Universal Robots URScript: Floor Corner Extended.script

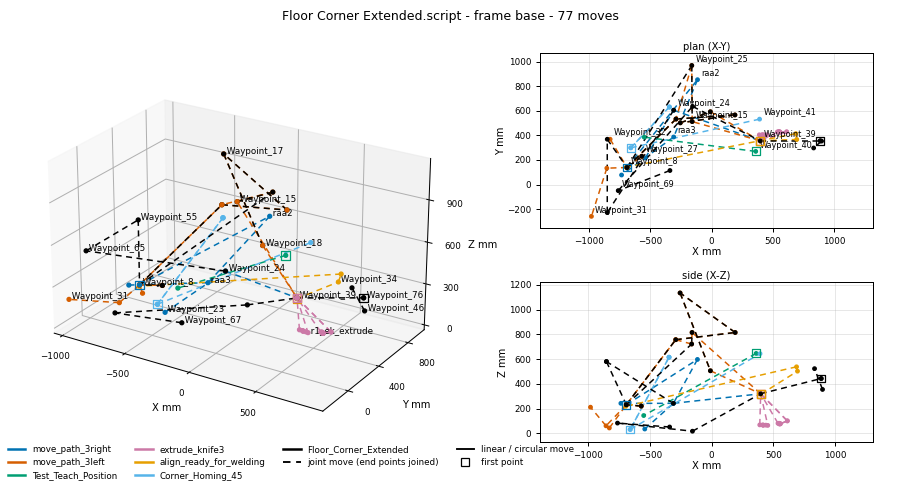
[picture p0: tool path of Floor Corner Extended.script in frame base, 77 of 152 moves have a stored position in this frame; points joined in program order, loops and branches not executed]
def Floor_Corner_Extended():
  global _hidden_verificationVariable=0
  step_count_477d2b75_14a1_4bd1_8ed8_9c73e5511d13 = 0.0
  thread Step_Counter_Thread_391a7927_408d_45dc_aa4e_0d8bac6dafc5():
    while (True):
      step_count_477d2b75_14a1_4bd1_8ed8_9c73e5511d13 = step_count_477d2b75_14a1_4bd1_8ed8_9c73e5511d13 + 1.0
      sync()
    end
  end
  run Step_Counter_Thread_391a7927_408d_45dc_aa4e_0d8bac6dafc5()
  set_tool_communication(False, 115200, 0, 1, 1.5, 3.5)
  set_tool_output_mode(0)
  set_tool_digital_output_mode(0, 1)
  set_tool_digital_output_mode(1, 1)
  set_tool_voltage(0)
  set_tcp(p[1.4000000000000001E-4,-0.01751,0.284,0.0,0.0,0.0])
  set_target_payload(10.800000, [-0.001000, -0.053000, 0.068000], [0.081228, 0.081228, 0.081228, 0.000000, 0.000000, 0.000000])
  set_gravity([0.0, 0.0, 9.82])
  set_standard_analog_input_domain(0, 1)
  set_standard_analog_input_domain(1, 1)
  set_tool_analog_input_domain(0, 1)
  set_tool_analog_input_domain(1, 1)
  set_analog_outputdomain(0, 0)
  set_analog_outputdomain(1, 0)
  set_input_actions_to_default()
  set_safety_mode_transition_hardness(1)
  global robot_number=2
  global Point_1=p[0.0,0.0,0.0,0.0,0.0,0.0]
  global Point_2=p[0.0,0.0,0.0,0.0,0.0,0.0]
  # begin: URCap Installation Node
  #   Source: UR Connect, 1.13.79, Universal Robots
  #   Type: UR Connect
  myurRPC = rpc_factory("xmlrpc","http://127.0.0.1:40474")
  # end: URCap Installation Node
  # begin: URCap Installation Node
  #   Source: MachineLogic for Universal Robots, 3.1.7, Vention Inc.
  #   Type: MachineLogic for Universal Robots
  def waitForResponse(expected_response_vention, cname_vention):
  response_vention = socket_read_string(cname_vention,timeout=15)
  while response_vention != expected_response_vention:
  sleep(0.01)
  response_vention = socket_read_string(cname_vention,timeout=15)
  end
  sleep(0.01)
  sync()
  end
  def sendString(string_vention, expected_response_vention, cname_vention):
  socket_send_string(str_cat(string_vention,";"), cname_vention)
  response_vention = socket_read_string(cname_vention,timeout=15)
  if(response_vention == "nAck"):
  popup("nAck received")
  end
  while response_vention != expected_response_vention:
  sleep(0.01)
  response_vention = socket_read_string(cname_vention,timeout=15)
  if(response_vention == "nAck"):
  popup("nAck received")
  end
  end
  sleep(0.01)
  sync()
  end
  def sendStringNAck(string_vention, expected_response_vention, cname_vention):
  socket_send_string(str_cat(string_vention,";"), cname_vention)
  response_vention = socket_read_string(cname_vention,timeout=15)
  if(response_vention == "nAck"):
  popup("nAck received")
  end
  while(response_vention != expected_response_vention and response_vention != "nAck"):
  sleep(0.01)
  response_vention = socket_read_string(cname_vention,timeout=15)
  if(response_vention == "nAck"):
  popup("nAck received",blocking=True)
  end
  end
  sleep(0.01)
  sync()
  end
  def sendStringWithTimeout(string_vention, expected_response_vention, cname_vention):
  socket_send_string(str_cat(string_vention,";"), cname_vention)
  response_vention = socket_read_string(cname_vention,timeout=10)
  if(response_vention == "nAck"):
  popup("nAck received"+string_vention)
  end
  sleep(0.01)
  sync()
  end
  def pollString(string_vention, expected_response_vention, cname_vention):
  socket_send_string(str_cat(string_vention,";"), cname_vention)
  response_vention = socket_read_string(cname_vention,timeout=15)
  if(response_vention == "nAck"):
  popup("nAck received")
  end
  while response_vention != expected_response_vention:
  sleep(1)
  socket_send_string(str_cat(string_vention,";"), cname_vention)
  response_vention = socket_read_string(cname_vention,timeout=15)
  if(response_vention == "nAck"):
  popup("nAck received")
  end
  end
  sleep(0.01)
  sync()
  end
  def sendVariable(var_vention, data_vention, expected_response_vention, cname_vention):
  socket_set_var(var_vention, data_vention, cname_vention)
  response_vention = socket_read_string(cname_vention,timeout=15)
  if(response_vention == "nAck"):
  popup("nAck received")
  end
  while response_vention != expected_response_vention:
  sleep(0.01)
  response_vention = socket_read_string(cname_vention,timeout=15)
  if(response_vention == "nAck"):
  popup("nAck received")
  end
  end
  sleep(0.01)
  sync()
  end
  def intToString(integer_vention,cname_vention):
  stringFix=""
  multiplier_vention123=1
  if integer_vention<0:
  stringFix="-"
  multiplier_vention123=-1
  end
  socket_set_var("GetString",integer_vention*multiplier_vention123,cname_vention)
  string_vention=""
  while string_vention=="":
  sleep(0.01)
  string_vention=socket_read_string(cname_vention,timeout=15)
  end
  sleep(0.01)
  sync()
  string_vention=stringFix+string_vention
  return string_vention
  end
  string_vention=""
  isVentionMovementBusy = False
  isVentionParallelMovementSendingScript = False
  ventionThreadHandle = 1
  isVentionMovementBusyMachineMotion1 = False
  isVentionParallelMovementSendingScriptMachineMotion1 = False
  socket_vention = socket_open("192.168.3.52", 9999, "MachineMotion1")
  if socket_vention==False:
  popup("Check configuration, can't connect to MachineMotion")
  end
  waitForResponse("MachineMotion connection established", "MachineMotion1")
  sendString("isReady", "MachineMotion isReady = true", "MachineMotion1")
  sendStringWithTimeout("setURCapVersion2", "setURCapVersion loaded", "MachineMotion1")
  sendString("SET speed_v2 1000000", "Ack", "MachineMotion1")
  sendString("SET acceleration_v2 100000", "Ack", "MachineMotion1")
  sendString("SET de_axis_1_microsteps_config 8", "Ack", "MachineMotion1")
  sendString("SET de_axis_1_mechanical_gain_config_v2 150000.0", "Ack", "MachineMotion1")
  sendString("SET de_axis_1_direction_config 1", "Ack", "MachineMotion1")
  sendString("SET de_axis_1_type_config Custom Actuator ", "Ack", "MachineMotion1")
  sendString("de_axis_1_config_exec", "Ack", "MachineMotion1")
  # end: URCap Installation Node
  # begin: URCap Installation Node
  #   Source: WireTank Serial, 4.9.0, WireTank, LLC
  #   Type: WireTank Serial
  WTSerialBridge = rpc_factory("xmlrpc","http://127.0.0.1:40511/RPC2")
  # end: URCap Installation Node
  global free_dr_already=  False
  global freedrive_m_var=  False
  global Waypoint_76_p=p[.886939072471, .356263001241, .442999104957, 2.316306590719, 2.057646408592, .074101958719]
  global Waypoint_76_q=[-3.2647881984118814, -1.2522049299371645, 1.5824044773896437, 0.9175786249801816, -0.008369636028316307, -1.3112608249927966]
  global Waypoint_50_p=p[-.568711442653, .230601791901, .220208834751, -1.519093932087, -.535128035721, .573965472012]
  global Waypoint_50_q=[-0.021522347127095998, -1.2794721287539979, 2.4323821703540247, 5.090870934515753, -2.2996109167682093, 1.533644199371338]
  global Waypoint_51_p=p[-.689649894186, .139001107022, .230693120258, -.852023156701, -1.645963115617, 1.645984943001]
  global Waypoint_51_q=[-1.1454814116107386, -1.5427037247321387, 2.8454700152026575, 4.979047852545538, -4.902958456669943, 1.5718834400177002]
  global Waypoint_52_p=p[-.160992057407, .970528182050, .722037363514, -.554955923310, .106486629259, .328544950173]
  global Waypoint_52_q=[-1.2978580633746546, -1.3217003357461472, 2.2583277861224573, 3.7025129038044433, -2.952825371419088, 0.9627944231033325]
  global Waypoint_53_p=p[-.157624488365, .513351401913, .815670293526, -.672704566373, -1.852329693545, -.055423312366]
  global Waypoint_53_q=[-2.7676661650287073, -1.8206430874266566, 2.312763277684347, 1.0122546392628173, -1.0765226523028772, -0.8102834860431116]
  global Waypoint_54_p=p[-.308528116178, .606080777007, .242371251996, -2.133736658076, .349438277129, 2.130953356703]
  global Waypoint_54_q=[-1.9617512861834925, -1.2994225782207032, 2.207935158406393, 0.745708628291748, 1.5955500602722168, 1.41863214969635]
  global Waypoint_65_p=p[-.850299549699, -.229060500451, .580194265918, -.066683564301, -1.566406749139, -.045536147896]
  global Waypoint_65_q=[0.11527767777442932, -1.206728772526123, 2.660132948552267, 3.2525827127644042, -4.69939905801882, -0.18521625200380498]
  global Waypoint_55_p=p[-.850295942693, .369353811615, .580190947871, -.066690142153, -1.566409865149, -.045506050424]
  global Waypoint_55_q=[-0.89636737505068, -1.198587493305542, 2.6061368624316614, 3.3119169908710937, -4.700617257748739, 0.826545238494873]
  global Waypoint_59_p=p[-.689650832419, .138973473550, .230700469426, -.851985360280, -1.645991124348, 1.645990580233]
  global Waypoint_59_q=[-1.1454528013812464, -1.5427289356342335, 2.8454795519458216, 4.979044186859884, -4.902960960065023, 1.5718833208084106]
  global Waypoint_71_p=p[-.289684660393, .534258475721, .757199031184, -.295236718653, -.653013693815, .389426431276]
  global Waypoint_71_q=[-1.3941848913775843, -1.6550847492613734, 2.7336130777942103, 4.156678839320801, -3.798194471989767, 1.7310842275619507]
  global Waypoint_58_p=p[.191120239889, .567518478899, .815512910186, -.135765364935, .396070873472, .208834263225]
  global Waypoint_58_q=[-1.651280705128805, -1.7712346516051234, 2.617981735860006, 3.3066598612019042, -2.656208101903097, 0.8563313484191895]
  global Waypoint_56_p=p[-.254568281661, .502958752129, 1.135400507516, -.261908057482, -.749714619963, 1.349050618455]
  global Waypoint_56_q=[-2.0344861189471644, -1.9012485943236292, 2.469647232686178, 2.2012061315723876, -1.1677187124835413, -0.5094392935382288]
  global Waypoint_57_p=p[-.009221327687, .593713365169, .505808930157, -1.424394189587, -2.344106819810, -.527597949261]
  global Waypoint_57_q=[-2.920837704335348, -1.9932075939574183, 2.3856611887561243, 0.6815890508839111, -0.5688460508929651, -1.1506975332843226]
  global Waypoint_67_p=p[-.339169194335, .114271165560, .051007401747, -.434162127311, 1.872717119498, -1.885153895998]
  global Waypoint_67_q=[-1.410516087208883, -0.9778240484050293, 2.47756010690798, -1.72361483196401, -0.3956816832171839, 1.808600902557373]
  global Waypoint_69_p=p[-.760826542313, -.049762698068, .082649581767, -1.026233921905, -1.612699318499, 1.547123897415]
  global Waypoint_69_q=[-0.22154647508730108, -1.118469015961029, 2.7561236063586634, -1.5568565337783475, -3.851987902318136, 1.559481143951416]
  global Waypoint_70_p=p[-.154414768496, .636923137577, .016979120256, -.302753655748, 1.486961848367, .122240024639]
  global Waypoint_70_q=[-1.1281922499286097, -1.0678585332683106, 2.4290812651263636, -2.7994214497008265, -1.6034835020648401, 1.7401196956634521]
  global Waypoint_49_p=p[.397354147848, .356263001249, .319808682466, 2.316306590727, 2.057646408591, .074101958728]
  global Waypoint_49_q=[-3.4579480330096644, -2.0568953953185023, 2.3266006151782435, -0.2270372670939942, -0.1993797461139124, -0.10534602800478154]
  global Waypoint_75_p=p[.886939072471, .356263001241, .442999104957, 2.316306590719, 2.057646408592, .074101958719]
  global Waypoint_75_q=[-3.2647881984118814, -1.2522049299371645, 1.5824044773896437, 0.9175786249801816, -0.008369636028316307, -1.3112608249927966]
  global Waypoint_46_p=p[.897631799353, .353934909904, .354805178378, 2.318109555057, 2.056931948624, .061383861333]
  global Waypoint_46_q=[-3.2637236754046843, -1.174605057840683, 1.6528332869159141, 1.0000695425220945, -0.0017340818988245132, -1.5358897417550086]
  global Waypoint_20_p=p[.833090611797, .298095916052, .522915034559, -2.069934341898, -1.817090229983, .262480162787]
  global Waypoint_20_q=[-3.3684676667627205, -1.191816195275802, 1.4015747865517827, 0.7519456332104983, -0.12742073350990069, -0.5504001287532203]
  global Waypoint_8_p=p[-.689650873132, .138963273545, .230691387978, -.851994598965, -1.645998530536, 1.646007616333]
  global Waypoint_8_q=[-0.9414032141314905, -1.501500443821289, 2.801856819783346, 4.981602895050802, -4.698942009602682, 1.571649193763733]
  global raa1_p=p[-.689643170661, .139073527807, .230690921608, -.852069296672, -1.645944888292, 1.645881185303]
  global raa1_q=[-1.1455705801593226, -1.5426994071206828, 2.8454588095294397, 4.979022520571508, -4.9029627482043665, 1.5718539953231812]
  global raa2_p=p[-.114157470946, .855108345894, .597477301975, -.505907028801, .325764798924, .388694870300]
  global raa2_q=[-1.2560303846942347, -1.339010552769043, 2.4151175657855433, 3.6540276247211914, -2.7377544085132044, 1.1360299587249756]
  global raa3_p=p[-.308547482234, .387797636904, .242407099860, 1.976327760240, .350206946999, -1.916000398832]
  global raa3_q=[-1.8931763807879847, -1.3096025747111817, 2.212959591542379, 0.7217818933674316, 1.639076590538025, 0.8125834465026855]
  global raa4_p=p[-.733576132099, .077690893520, .242409727900, 1.976419296976, .350069431278, -1.916084616091]
  global raa4_q=[-0.8909156958209437, -1.3431089532426377, 2.273750130330221, 0.7266384798237304, 1.5611975193023682, 1.8127720355987549]
  global Waypoint_23_p=p[-.540166575654, .215949141041, .034631452617, -1.505795438113, 1.057579835594, 1.573514753692]
  global Waypoint_23_q=[-0.46167117754091436, -1.1365486842444916, 2.508885685597555, 0.15223841249432368, 1.4952874183654785, 3.819530963897705]
  global Waypoint_24_p=p[-.308525559537, .606096497354, .242373144855, -2.133742737559, .349425192770, 2.130939839044]
  global Waypoint_24_q=[-1.8709262053119105, -1.2877716285041352, 2.192875687276022, 0.7510036665150146, 1.5878156423568726, 1.5091480016708374]
  global Waypoint_39_p=p[.397377312153, .356253310648, .319810281486, 2.316317670744, 2.057592854035, .074120023159]
  global Waypoint_39_q=[-3.4579551855670374, -2.0568958721556605, 2.3265963236438196, -0.22706706941638188, -0.19935590425600225, -0.10534030595888311]
  global Waypoint_37_p=p[.397366630181, .356258644196, .319813668943, 2.316299214281, 2.057614642521, .074125657910]
  global Waypoint_37_q=[-3.4579508940326136, -2.056904455224508, 2.3265963236438196, -0.2270481151393433, -0.19937020937074834, -0.10535222688783819]
  global Waypoint_15_p=p[-.157621040248, .513353603496, .815677694745, -.672699538592, -1.852318447516, -.055422773001]
  global Waypoint_15_q=[-2.770456854497091, -1.8207680187621058, 2.3065691629992884, 1.0170823770710449, -1.0767205397235315, -0.8071182409869593]
  global Waypoint_25_p=p[-.161036555831, .970524399959, .722042384791, -.554954311189, .106465018540, .328580879483]
  global Waypoint_25_q=[-1.3071630636798304, -1.3366777312806626, 2.2083633581744593, 3.7187773424335937, -2.9519384543048304, 0.9132363796234131]
  global Waypoint_72_p=p[-.289685725237, .534256396594, .757196155975, -.295237726329, -.653009715205, .389435972469]
  global Waypoint_72_q=[-1.394179646168844, -1.6550847492613734, 2.7336154619800013, 4.156686468715332, -3.7981911341296595, 1.731092095375061]
  global Waypoint_26_p=p[-.689650873132, .138963273545, .230691387978, -.851994598965, -1.645998530536, 1.646007616333]
  global Waypoint_26_q=[-0.9414032141314905, -1.501500443821289, 2.801856819783346, 4.981602895050802, -4.698942009602682, 1.571649193763733]
  global Waypoint_27_p=p[-.568724745609, .230601805298, .220208295176, -1.519097711196, -.535155391172, .573964121010]
  global Waypoint_27_q=[-0.04883271852602178, -1.2753942471793671, 2.4771457354175013, 5.041022258787908, -2.326899592076437, 1.532160997390747]
  global Waypoint_28_p=p[-.568724745609, .230601805298, .220208295176, -1.519097711196, -.535155391172, .573964121010]
  global Waypoint_28_q=[-0.04883271852602178, -1.2753942471793671, 2.4771457354175013, 5.041022258787908, -2.326899592076437, 1.532160997390747]
  global Waypoint_29_p=p[-.689650873132, .138963273545, .230691387978, -.851994598965, -1.645998530536, 1.646007616333]
  global Waypoint_29_q=[-0.9414032141314905, -1.501500443821289, 2.801856819783346, 4.981602895050802, -4.698942009602682, 1.571649193763733]
  global Waypoint_30_p=p[-.853851193668, .133266829906, .060418082908, -.274178222953, -2.359710051999, .046821166283]
  global Waypoint_30_q=[-0.608560864125387, -1.0122360748103638, 2.787060801182882, 3.7283646303364257, -4.940747324620382, 0.3777344226837158]
  global Waypoint_31_p=p[-.979398188272, -.259625449453, .211289397035, -.673010443572, -1.459355862765, -.640164958946]
  global Waypoint_31_q=[0.36968713998794556, -0.5732358259013672, 2.138303581868307, 3.1253925996967773, -4.70385724702944, -1.2100523153888147]
  global Waypoint_32_p=p[-.826865752305, .369357632284, .043113676955, .574997346548, -1.492225541214, .597128135378]
  global Waypoint_32_q=[-1.0355513731585901, -0.33930082738909917, 2.126244846974508, 2.9386045175739746, -4.711197797452108, 1.7860286235809326]
  global Waypoint_33_p=p[-.689650873132, .138963273545, .230691387978, -.851994598965, -1.645998530536, 1.646007616333]
  global Waypoint_33_q=[-0.9414032141314905, -1.501500443821289, 2.801856819783346, 4.981602895050802, -4.698942009602682, 1.571649193763733]
  global Waypoint_73_p=p[-.289671192632, .534275423553, .757232902417, -.295189983811, -.652980753171, .389398176275]
  global Waypoint_73_q=[-1.39418870607485, -1.65509094814443, 2.7335642019854944, 4.156684561366699, -3.7981610933886927, 1.731088399887085]
  global Waypoint_16_p=p[.191112811238, .567512170908, .815514010937, -.135771161622, .396053809900, .208825693369]
  global Waypoint_16_q=[-1.6536315123187464, -1.762029310266012, 2.6225650946246546, 3.2891055780598144, -2.6549678484546106, 0.8520665764808655]
  global Waypoint_17_p=p[-.254565633623, .502963426820, 1.135401557820, -.261910507478, -.749716086887, 1.349041636154]
  global Waypoint_17_q=[-2.035229508076803, -1.8928028545775355, 2.468372408543722, 2.19391576826062, -1.167032543812887, -0.5091407934771937]
  global Waypoint_18_p=p[-.009208376822, .593717720951, .505810027228, -1.424406033077, -2.344120510145, -.527630245278]
  global Waypoint_18_q=[-2.9172328154193323, -1.9945279560484828, 2.3804522196399134, 0.6930715280720214, -0.5671199003802698, -1.1566088835345667]
  global Waypoint_38_p=p[.397379749540, .356252016937, .319817140705, 2.316310534508, 2.057580214841, .074134378577]
  global Waypoint_38_q=[-3.457958761845724, -2.0569073162474574, 2.3265913168536585, -0.22705944002185063, -0.19935638109316045, -0.10534793535341436]
  global Waypoint_40_p=p[.360688403366, .270119715397, .646144746546, .057805349154, 2.125995180379, 2.134053153683]
  global Waypoint_40_q=[-3.4579489866839808, -2.0569035015501917, 2.3265796343432825, -0.22706706941638188, -0.1993501822101038, -0.10534793535341436]
  global Waypoint_2_p=p[-.548957282596, .386284559177, .143710178207, 1.570800598292, -.000025190822, .000004803470]
  global Waypoint_2_q=[-1.0516188780414026, -1.010990933781006, 2.1562450567828577, -1.143702046280243, -1.0526168982135218, -0.0017235914813440445]
  global r1_ek_oldhome_p=p[.397380247322, .356253634699, .319820846021, 2.316316320871, 2.057594704604, .074118471609]
  global r1_ek_oldhome_q=[-3.457949940358297, -2.056894441644186, 2.32658034959902, -0.2270551484874268, -0.19935208955873662, -0.10533696809877569]
  global r1_ek_extrude_p=p[.454852104155, .405448828659, .064015413765, 2.316807606413, 2.051392071696, .076664825947]
  global r1_ek_extrude_q=[-3.274653975163595, -1.5604325172356148, 2.467809502278463, -0.34438879907641606, -0.014281574879781544, -0.6303489843951624]
  global r1_ek_front_p=p[.439064809878, .405452261046, .065996139932, 2.316843937268, 2.051427632497, .076607106393]
  global r1_ek_front_q=[-3.280560557042257, -1.6287623844542445, 2.502561871205465, -0.47416289270434575, -0.019731823598043263, -0.4669149557696741]
  global r1_ek_middle_p=p[.419010105608, .404850828431, .065994665459, 2.309574128677, 2.044678176343, .089098333896]
  global r1_ek_middle_q=[-3.290863100682394, -1.70143522838735, 2.548208538685934, -0.589385525589325, -0.029501263295308888, -0.3372734228717249]
  global r1_ek_middle2_p=p[.417011768852, .405435328663, .065002627117, 2.316867113472, 2.051334925313, .076628493429]
  global r1_ek_middle2_q=[-3.289830032979147, -1.6934038601317347, 2.5445857683764856, -0.579618052845337, -0.028589550648824513, -0.33885270753969365]
  global r1_ek_bottom_p=p[.413071667620, .405431286494, .067999701073, 2.316819721954, 2.051304037200, .076688572349]
  global r1_ek_bottom_q=[-3.2916205565081995, -1.708447118798727, 2.5485368410693567, -0.5849895042232056, -0.03033763567079717, -0.32244998613466436]
  global r1_ek_end_p=p[.389998638281, .405443674081, .068004818811, 2.316851991921, 2.051367741778, .076612018685]
  global r1_ek_end_q=[-3.3030064741717737, -1.7640062771239222, 2.5831297079669397, -0.63420523822818, -0.04154044786562139, -0.2521465460406702]
  global r2_ek_oldhome_p=p[.397380247322, .356253634699, .319820846021, 2.316316320871, 2.057594704604, .074118471609]
  global r2_ek_oldhome_q=[-3.461132842686933, -2.062320779349874, 2.32916033290004, -0.21924456446492258, -0.20097883707844666, -0.11039879152527199]
  global r2_ek_extrude_p=p[.612885745678, .429305279732, .100477107124, 2.149994969793, 2.225764025207, .087353352584]
  global r2_ek_extrude_q=[-3.199475796455825, -1.4862854517875999, 2.263543898005424, -0.6928175084157413, -0.09183293866530295, -0.15653548683830643]
  global r2_ek_front_p=p[.556405415915, .429305279815, .076984362723, -2.170411249256, -2.268200695165, -.015853660170]
  global r2_ek_front_q=[-3.2029012478485694, -1.4943971905029905, 2.3176866046272355, -0.727203417516419, -0.10461513056100813, -0.1013922369747533]
  global r2_ek_middle_p=p[.550033970532, .429305279917, .076253920653, -2.170411249261, -2.268200695170, -.015853660159]
  global r2_ek_middle_q=[-3.2036200175167613, -1.5006788185274456, 2.326226188945654, -0.730095076239345, -0.10533288811000929, -0.10075548926859312]
  global r2_ek_bottom_p=p[.546594660555, .429305280025, .080868477599, -2.170411249265, -2.268200695174, -.015853660149]
  global r2_ek_bottom_q=[-3.204010221105431, -1.5099366263094405, 2.3272215014458872, -0.722096275899732, -0.10572512264357048, -0.10049057923478166]
  global r2_ek_end_p=p[.537335106646, .429305280055, .080868477459, -2.170411249266, -2.268200695175, -.015853660146]
  global r2_ek_end_q=[-3.205098875769389, -1.5204959829395506, 2.3387656715508855, -0.724001524008818, -0.10681294496314919, -0.09956563917089412]
  global oldhome_p=p[.397683836105, .356251384911, .315246899233, 2.316304177919, 2.057561756051, .074146544723]
  global oldhome_q=[-3.457960907612936, -2.0569125614561976, 2.326589886342184, -0.22707636774096684, -0.19935208955873662, -0.10534269014467412]
  global Waypoint_34_p=p[.695155464390, .367451880816, .502522491683, 2.093108370749, 1.857548644474, .308841595089]
  global Waypoint_34_q=[-3.249415699635641, -1.9387923679747523, 2.3226097265826624, 3.981850786800049, -0.05697328249086553, 1.5286790132522583]
  global Waypoint_35_p=p[.687527620967, .415165960724, .537921070000, 2.127101811831, 1.929915403723, .470130777221]
  global Waypoint_35_q=[-3.249424997960226, -1.9387947521605433, 2.32263428369631, 3.9818588930317382, -6.198007937763826, 1.5286580324172974]
  global Waypoint_36_p=p[-.693756081485, .141369193308, .218584735520, -.851978179689, -1.646001533937, 1.646008371360]
  global Waypoint_36_q=[-1.1533568541156214, -1.4924076360515137, 2.8518698851214808, 4.922323781042852, -4.910887185727255, 1.5719373226165771]
  def calculate_point_to_move_towards(feature, direction, position_distance):
    local posDir=[direction[0], direction[1], direction[2]]
    if (norm(posDir) < 1e-6):
      return get_target_waypoint()
    end
    local direction_vector_normalized=normalize(posDir)
    local displacement_pose=p[direction_vector_normalized[0] * position_distance,direction_vector_normalized[1] * position_distance,direction_vector_normalized[2] * position_distance,0,0,0]
    local wanted_displacement_in_base_frame=pose_sub(pose_trans(feature, displacement_pose), feature)
    return pose_add(get_target_waypoint(), wanted_displacement_in_base_frame)
  end
  global Waypoint_4_p=p[-.658264763546, .299530128456, .030909835036, .426821001551, -1.621505068649, .437070885767]
  global Waypoint_4_q=[-1.350241486226217, -0.9702387017062684, 2.492185179387228, -1.7834822140135707, -0.33723670641054326, 1.8489984273910522]
  global Waypoint_13_p=p[-.343952006273, .632142227752, .615174722549, -.025948978133, -.008794819136, -.567469912202]
  global Waypoint_13_q=[-1.350241486226217, -0.9702451390079041, 2.492171827946798, -3.0669099293150843, 1.575993537902832, 2.355180025100708]
  global Waypoint_1_p=p[-.343952006258, .632142227456, .615174722551, -.025016780489, .033118613186, -3.068519793995]
  global Waypoint_1_q=[-1.3432858302651205, -0.8819789687502322, 2.478150442072055, -3.1920490209023007, 1.5816449765089289, -0.1549241290366341]
  global Waypoint_14_p=p[-.343952006273, .632142227752, .615174722549, -.025948978133, -.008794819136, -.567469912202]
  global Waypoint_14_q=[-1.350241486226217, -0.9702451390079041, 2.492171827946798, -3.0669099293150843, 1.575993537902832, 2.355180025100708]
  global Waypoint_41_p=p[.392127936214, .533269017847, .644148583936, .057822570580, 2.125982462550, 2.134033989912]
  global Waypoint_41_q=[-3.4579578081714075, -2.0569120846190394, 2.3265841642962855, -0.22706885755572515, -0.1993349234210413, -0.10534984270204717]
  def move_path_3right():
    $ 136 "move_path_3right" "noBreak"
    $ 137 "'this is the path for Down, Over, then Back Around'"
    # 'this is the path for Down, Over, then Back Around'
    $ 138 "Comment"
    # Comment
    $ 147 "align_ready_for_welding()"
    align_ready_for_welding()
    $ 148 "Comment"
    # Comment
    $ 149 "Set"
    set_tcp(p[-0.011699999999999999,-0.328,0.105,1.2092,-1.2092,1.2092])
    $ 150 "p1≔pathturn[0]"
    global p1=pathturn[0]
    $ 151 "p2≔pathturn[1]"
    global p2=pathturn[1]
    $ 152 "p4≔pathturn[2]"
    global p4=pathturn[2]
    $ 153 "p5≔pathturn[3]"
    global p5=pathturn[3]
    $ 154 "pa1≔p[p1[0]+0.05,p1[1]+0.05,p1[2],p1[3],p1[4],p1[5]]"
    global pa1=p[p1[0]+0.05,p1[1]+0.05,p1[2],p1[3],p1[4],p1[5]]
    $ 155 "liftcolumnup"
    $ 156 "liftcolumnz≔liftcolumnzneeded"
    global liftcolumnz=liftcolumnzneeded
    $ 157 "If liftcolumnz>0"
    if (liftcolumnz>0):
      # begin: URCap Program Node
      #   Source: MachineLogic for Universal Robots, 3.1.7, Vention Inc.
      #   Type: MachineLogic for Universal Robots
      $ 158 "MachineLogic Move to Position"
      while isVentionMovementBusyMachineMotion1==True:
      sleep(0.05)
      end
      if(isVentionMovementBusyMachineMotion1 == False):
      isVentionMovementBusyMachineMotion1 = True
      socket_send_string("estop/status;", "MachineMotion1")
      temp_estop_var_vention = socket_read_string("MachineMotion1",timeout=15)
      while(temp_estop_var_vention=="estop/status true"):
      if temp_estop_var_vention=="estop/status true":
      sendStringWithTimeout("estop/systemreset/request","Ack estop/systemreset/request;","MachineMotion1")
      end
      socket_send_string("estop/status;", "MachineMotion1")
      temp_estop_var_vention = socket_read_string("MachineMotion1",timeout=15)
      if temp_estop_var_vention=="estop/status true":
      popup("MachineMotion in estop, make sure you have all emergency modules released manually. If you continue the system will try to reset MachineMotion automatically.",blocking=True)
      end
      end
      else:
      popup("resource is being used already: MachineMotion1")
      halt
      end
      sendString("SET speed_v2 3000000.000", "Ack", "MachineMotion1")
      sendString("SET acceleration_v2 50000.000", "Ack", "MachineMotion1")
      string_vention=intToString(liftcolumnz*1000,"MachineMotion1")
      sendString("SET de_move_abs_1 "+string_vention, "Ack", "MachineMotion1")
      sendString("de_move_abs_exec", "Ack", "MachineMotion1")
      isVentionParallelMovementSendingScriptMachineMotion1 = False
      pollString("isMotionCompleted", "MachineMotion isMotionCompleted = true", "MachineMotion1")
      isVentionMovementBusyMachineMotion1 = False
      sleep(0.03)
      # end: URCap Program Node
    end
    $ 159 "MoveJ"
    $ 160 "pa1" "breakAfter"
    movej(pa1, a=1.3962634015954636, v=0.3490658503988659)
    $ 161 "MoveL"
    $ 162 "p1" "breakAfter"
    movel(p1, a=0.2, v=0.05)
    $ 163 "Wait: 8.0"
    sleep(8.0)
    # begin: URCap Program Node
    #   Source: WireTank Serial, 4.9.0, WireTank, LLC
    #   Type: WireTank Serial
    $ 164 "Serial Bridge uR1"
    SerialResponse = WTSerialBridge.send_command("/dev/ttyUSB0",1200, 8, "None", "One", "None", 1000, "None", "None", [252,82,49], False)
    # end: URCap Program Node
    # begin: URCap Program Node
    #   Source: WireTank Serial, 4.9.0, WireTank, LLC
    #   Type: WireTank Serial
    $ 165 "Serial Bridge uR1"
    SerialResponse = WTSerialBridge.send_command("/dev/ttyUSB0",1200, 8, "None", "One", "None", 1000, "None", "None", [252,82,49], False)
    # end: URCap Program Node
    $ 166 "Wait: 1.0"
    sleep(1.0)
    $ 168 "Set DO[0]=On"
    set_standard_digital_out(0, True)
    $ 169 "MoveL"
    $ 170 "p2" "breakAfter"
    movel(p2, a=0.1, v=0.01)
    # begin: URCap Program Node
    #   Source: WireTank Serial, 4.9.0, WireTank, LLC
    #   Type: WireTank Serial
    $ 171 "Serial Bridge uR0"
    SerialResponse = WTSerialBridge.send_command("/dev/ttyUSB0",1200, 8, "None", "One", "None", 1000, "None", "None", [252,82,48], False)
    # end: URCap Program Node
    $ 172 "Wait: 0.5"
    sleep(0.5)
    $ 173 "Set DO[0]=Off"
    set_standard_digital_out(0, False)
    $ 174 "MoveL"
    $ 175 "p4" "breakAfter"
    movel(p4, a=0.01, v=0.12)
    # begin: URCap Program Node
    #   Source: WireTank Serial, 4.9.0, WireTank, LLC
    #   Type: WireTank Serial
    $ 176 "Serial Bridge uR1"
    SerialResponse = WTSerialBridge.send_command("/dev/ttyUSB0",1200, 8, "None", "One", "None", 1000, "None", "None", [252,82,49], False)
    # end: URCap Program Node
    # begin: URCap Program Node
    #   Source: WireTank Serial, 4.9.0, WireTank, LLC
    #   Type: WireTank Serial
    $ 177 "Serial Bridge uR1"
    SerialResponse = WTSerialBridge.send_command("/dev/ttyUSB0",1200, 8, "None", "One", "None", 1000, "None", "None", [252,82,49], False)
    # end: URCap Program Node
    $ 178 "Wait: 1.0"
    sleep(1.0)
    $ 180 "Set DO[0]=On"
    set_standard_digital_out(0, True)
    $ 181 "MoveL"
    $ 182 "p5" "breakAfter"
    movel(p5, a=0.1, v=0.01)
    # begin: URCap Program Node
    #   Source: WireTank Serial, 4.9.0, WireTank, LLC
    #   Type: WireTank Serial
    $ 183 "Serial Bridge uR0"
    SerialResponse = WTSerialBridge.send_command("/dev/ttyUSB0",1200, 8, "None", "One", "None", 1000, "None", "None", [252,82,48], False)
    # end: URCap Program Node
    $ 184 "Wait: 2.0"
    sleep(2.0)
    $ 185 "Set DO[0]=Off"
    set_standard_digital_out(0, False)
    $ 186 "Comment"
    # Comment
    $ 187 "pret1≔p[p5[0]+.1,p5[1],p5[2],p5[3],p5[4],p5[5]]"
    global pret1=p[p5[0]+.1,p5[1],p5[2],p5[3],p5[4],p5[5]]
    $ 188 "p_1≔pathturn[4]"
    global p_1=pathturn[4]
    $ 189 "p_2≔pathturn[5]"
    global p_2=pathturn[5]
    $ 190 "p_3≔pathturn[6]"
    global p_3=pathturn[6]
    $ 191 "p_4≔pathturn[7]"
    global p_4=pathturn[7]
    $ 192 "p_5≔pathturn[8]"
    global p_5=pathturn[8]
    $ 193 "p_preheat≔p[p_3[0]+.01,p_3[1],p_3[2],p_3[3],p_3[4],p_3[5]]"
    global p_preheat=p[p_3[0]+.01,p_3[1],p_3[2],p_3[3],p_3[4],p_3[5]]
    $ 194 "p_pre_ret≔p[p_1[0]+.03,p_1[1]+.03,p_1[2],p_1[3],p_1[4],p_1[5]]"
    global p_pre_ret=p[p_1[0]+.03,p_1[1]+.03,p_1[2],p_1[3],p_1[4],p_1[5]]
    $ 195 "p_pre_ret2≔p[p_3[0]+.1,p_3[1],p_3[2],p_3[3],p_3[4],p_3[5]]"
    global p_pre_ret2=p[p_3[0]+.1,p_3[1],p_3[2],p_3[3],p_3[4],p_3[5]]
    $ 196 "'twist'"
    # 'twist'
    $ 197 "MoveJ"
    $ 198 "pret1" "breakAfter"
    movej(pret1, a=1.3962634015954636, v=1.3962634015954636)
    $ 199 "Waypoint_8" "breakAfter"
    movej(get_inverse_kin(Waypoint_8_p, qnear=Waypoint_8_q), a=1.3962634015954636, v=1.0471975511965976)
    $ 201 "MoveJ"
    $ 202 "raa1" "breakAfter"
    movej(get_inverse_kin(raa1_p, qnear=raa1_q), a=1.3962634015954636, v=1.0471975511965976)
    $ 203 "raa2" "breakAfter"
    movej(get_inverse_kin(raa2_p, qnear=raa2_q), a=1.3962634015954636, v=1.0471975511965976)
    $ 204 "raa3" "breakAfter"
    movej(get_inverse_kin(raa3_p, qnear=raa3_q), a=1.3962634015954636, v=1.0471975511965976)
    $ 205 "raa4" "breakAfter"
    movej(get_inverse_kin(raa4_p, qnear=raa4_q), a=1.3962634015954636, v=1.0471975511965976)
    $ 207 "If liftcolumnz≠0.0"
    if (liftcolumnz != 0.0):
      # begin: URCap Program Node
      #   Source: MachineLogic for Universal Robots, 3.1.7, Vention Inc.
      #   Type: MachineLogic for Universal Robots
      $ 208 "MachineLogic Homing"
      while isVentionMovementBusyMachineMotion1==True:
      sleep(0.05)
      end
      if(isVentionMovementBusyMachineMotion1 == False):
      isVentionMovementBusyMachineMotion1 = True
      socket_send_string("estop/status;", "MachineMotion1")
      temp_estop_var_vention = socket_read_string("MachineMotion1",timeout=15)
      while(temp_estop_var_vention=="estop/status true"):
      if temp_estop_var_vention=="estop/status true":
      sendStringWithTimeout("estop/systemreset/request","Ack estop/systemreset/request;","MachineMotion1")
      end
      socket_send_string("estop/status;", "MachineMotion1")
      temp_estop_var_vention = socket_read_string("MachineMotion1",timeout=15)
      if temp_estop_var_vention=="estop/status true":
      popup("MachineMotion in estop, make sure you have all emergency modules released manually. If you continue the system will try to reset MachineMotion automatically.",blocking=True)
      end
      end
      else:
      popup("resource is being used already: MachineMotion1")
      halt
      end
      isVentionMovementBusyMachineMotion1 = True
      sendString("im_home_axis_1", "MachineMotion im_home_axis_1 = completed", "MachineMotion1")
      isVentionMovementBusyMachineMotion1 = False
      sendString("SET im_set_encoder_pos_aux_1 0.000", "Ack", "MachineMotion1")
      isVentionMovementBusyMachineMotion1 = False
      sleep(0.03)
      # end: URCap Program Node
    end
    $ 209 "'preheat'"
    # 'preheat'
    $ 212 "MoveL"
    $ 213 "p_pre_ret2" "breakAfter"
    movel(p_pre_ret2, a=1.2, v=0.25)
    $ 214 "p_preheat" "breakAfter"
    movel(p_preheat, a=1.2, v=0.25)
    $ 215 "Wait: 6.0"
    sleep(6.0)
    $ 216 "MoveL"
    $ 217 "p_pre_ret2" "breakAfter"
    movel(p_pre_ret2, a=1.2, v=0.25)
    $ 218 "p_pre_ret" "breakAfter"
    movel(p_pre_ret, a=1.2, v=0.25)
    $ 219 "Set"
    set_tcp(p[0.00451,-0.328,0.105,1.2092,-1.2092,1.2092])
    $ 220 "MoveL"
    $ 221 "p_1" "breakAfter"
    movel(p_1, a=1.2, v=0.05)
    # begin: URCap Program Node
    #   Source: WireTank Serial, 4.9.0, WireTank, LLC
    #   Type: WireTank Serial
    $ 222 "Serial Bridge uR1"
    SerialResponse = WTSerialBridge.send_command("/dev/ttyUSB0",1200, 8, "None", "One", "None", 1000, "None", "None", [252,82,49], False)
    # end: URCap Program Node
    # begin: URCap Program Node
    #   Source: WireTank Serial, 4.9.0, WireTank, LLC
    #   Type: WireTank Serial
    $ 223 "Serial Bridge uR1"
    SerialResponse = WTSerialBridge.send_command("/dev/ttyUSB0",1200, 8, "None", "One", "None", 1000, "None", "None", [252,82,49], False)
    # end: URCap Program Node
    $ 224 "Wait: 1.0"
    sleep(1.0)
    $ 225 "Set DO[0]=On"
    set_standard_digital_out(0, True)
    $ 227 "Wait: 1.0"
    sleep(1.0)
    $ 228 "MoveL"
    $ 229 "p_2" "breakAfter"
    movel(p_2, a=1.2, v=0.01)
    $ 230 "MoveP"
    $ 231 "CircleMove"
    $ 232 "p_3" "noBreak"

    $ 233 "p_4" "breakAfter"
    movec(p_3, p_4, a=0.01, v=5.0E-4, r=0.0, mode=1)
    $ 234 "MoveL"
    $ 235 "p_5" "breakAfter"
    movel(p_5, a=1.2, v=0.012)
    # begin: URCap Program Node
    #   Source: WireTank Serial, 4.9.0, WireTank, LLC
    #   Type: WireTank Serial
    $ 236 "Serial Bridge uR0"
    SerialResponse = WTSerialBridge.send_command("/dev/ttyUSB0",1200, 8, "None", "One", "None", 1000, "None", "None", [252,82,48], False)
    # end: URCap Program Node
    $ 237 "Wait: 2.0"
    sleep(2.0)
    $ 238 "Set DO[0]=Off"
    set_standard_digital_out(0, False)
    $ 239 "MoveL"
    $ 240 "Waypoint_23" "breakAfter"
    movel(Waypoint_23_p, a=1.2, v=0.25)
    $ 241 "MoveJ"
    $ 242 "Waypoint_24" "breakAfter"
    movej(get_inverse_kin(Waypoint_24_p, qnear=Waypoint_24_q), a=1.3962634015954636, v=1.0471975511965976)
    $ 243 "Waypoint_39" "breakAfter"
    movej(get_inverse_kin(Waypoint_39_p, qnear=Waypoint_39_q), a=1.3962634015954636, v=1.0471975511965976)
    $ 244 "'above waypoint is home'"
    # 'above waypoint is home'
  end
  def move_path_3left():
    $ 245 "move_path_3left" "noBreak"
    $ 246 "'this is the path for Down, Over, then Back Around'"
    # 'this is the path for Down, Over, then Back Around'
    $ 247 "Comment"
    # Comment
    $ 248 "MoveJ"
    $ 249 "Waypoint_37" "breakAfter"
    movej(get_inverse_kin(Waypoint_37_p, qnear=Waypoint_37_q), a=1.3962634015954636, v=1.0471975511965976)
    $ 250 "'above point is home'"
    # 'above point is home'
    $ 251 "liftcolumnup"
    $ 252 "liftcolumnz≔liftcolumnzneeded"
    global liftcolumnz=liftcolumnzneeded
    $ 253 "If liftcolumnz>0"
    if (liftcolumnz>0):
      # begin: URCap Program Node
      #   Source: MachineLogic for Universal Robots, 3.1.7, Vention Inc.
      #   Type: MachineLogic for Universal Robots
      $ 254 "MachineLogic Move to Position"
      while isVentionMovementBusyMachineMotion1==True:
      sleep(0.05)
      end
      if(isVentionMovementBusyMachineMotion1 == False):
      isVentionMovementBusyMachineMotion1 = True
      socket_send_string("estop/status;", "MachineMotion1")
      temp_estop_var_vention = socket_read_string("MachineMotion1",timeout=15)
      while(temp_estop_var_vention=="estop/status true"):
      if temp_estop_var_vention=="estop/status true":
      sendStringWithTimeout("estop/systemreset/request","Ack estop/systemreset/request;","MachineMotion1")
      end
      socket_send_string("estop/status;", "MachineMotion1")
      temp_estop_var_vention = socket_read_string("MachineMotion1",timeout=15)
      if temp_estop_var_vention=="estop/status true":
      popup("MachineMotion in estop, make sure you have all emergency modules released manually. If you continue the system will try to reset MachineMotion automatically.",blocking=True)
      end
      end
      else:
      popup("resource is being used already: MachineMotion1")
      halt
      end
      sendString("SET speed_v2 3000000.000", "Ack", "MachineMotion1")
      sendString("SET acceleration_v2 50000.000", "Ack", "MachineMotion1")
      string_vention=intToString(liftcolumnz*1000,"MachineMotion1")
      sendString("SET de_move_abs_1 "+string_vention, "Ack", "MachineMotion1")
      sendString("de_move_abs_exec", "Ack", "MachineMotion1")
      isVentionParallelMovementSendingScriptMachineMotion1 = False
      pollString("isMotionCompleted", "MachineMotion isMotionCompleted = true", "MachineMotion1")
      isVentionMovementBusyMachineMotion1 = False
      sleep(0.03)
      # end: URCap Program Node
    end
    $ 255 "Waypoint_15" "breakAfter"
    movej(get_inverse_kin(Waypoint_15_p, qnear=Waypoint_15_q), a=1.3962634015954636, v=1.0471975511965976)
    $ 256 "Waypoint_25" "breakAfter"
    movej(get_inverse_kin(Waypoint_25_p, qnear=Waypoint_25_q), a=1.3962634015954636, v=1.0471975511965976)
    $ 257 "Waypoint_72" "breakAfter"
    movej(get_inverse_kin(Waypoint_72_p, qnear=Waypoint_72_q), a=1.3962634015954636, v=1.0471975511965976)
    $ 258 "Waypoint_26" "breakAfter"
    movej(get_inverse_kin(Waypoint_26_p, qnear=Waypoint_26_q), a=1.3962634015954636, v=1.0471975511965976)
    $ 259 "Waypoint_27" "breakAfter"
    movej(get_inverse_kin(Waypoint_27_p, qnear=Waypoint_27_q), a=1.3962634015954636, v=1.0471975511965976)
    $ 264 "Comment"
    # Comment
    $ 265 "Set"
    set_tcp(p[-0.011699999999999999,-0.328,0.105,1.2092,-1.2092,1.2092])
    $ 266 "p1≔pathturn[0]"
    global p1=pathturn[0]
    $ 267 "p2≔pathturn[1]"
    global p2=pathturn[1]
    $ 268 "p4≔pathturn[2]"
    global p4=pathturn[2]
    $ 269 "p5≔pathturn[3]"
    global p5=pathturn[3]
    $ 270 "pa1≔p[p1[0]+0.05,p1[1]-0.05,p1[2],p1[3],p1[4],p1[5]]"
    global pa1=p[p1[0]+0.05,p1[1]-0.05,p1[2],p1[3],p1[4],p1[5]]
    $ 271 "MoveJ"
    $ 272 "pa1" "breakAfter"
    movej(pa1, a=1.3962634015954636, v=1.0471975511965976)
    $ 273 "MoveL"
    $ 274 "p1" "breakAfter"
    movel(p1, a=0.1, v=0.05)
    $ 275 "Wait: 8.0"
    sleep(8.0)
    # begin: URCap Program Node
    #   Source: WireTank Serial, 4.9.0, WireTank, LLC
    #   Type: WireTank Serial
    $ 276 "Serial Bridge uR1"
    SerialResponse = WTSerialBridge.send_command("/dev/ttyUSB0",1200, 8, "None", "One", "None", 1000, "None", "None", [252,82,49], False)
    # end: URCap Program Node
    # begin: URCap Program Node
    #   Source: WireTank Serial, 4.9.0, WireTank, LLC
    #   Type: WireTank Serial
    $ 277 "Serial Bridge uR1"
    SerialResponse = WTSerialBridge.send_command("/dev/ttyUSB0",1200, 8, "None", "One", "None", 1000, "None", "None", [252,82,49], False)
    # end: URCap Program Node
    $ 278 "Wait: 1.0"
    sleep(1.0)
    $ 280 "Set DO[0]=On"
    set_standard_digital_out(0, True)
    $ 281 "MoveL"
    $ 282 "p2" "breakAfter"
    movel(p2, a=0.1, v=0.01)
    # begin: URCap Program Node
    #   Source: WireTank Serial, 4.9.0, WireTank, LLC
    #   Type: WireTank Serial
    $ 283 "Serial Bridge uR0"
    SerialResponse = WTSerialBridge.send_command("/dev/ttyUSB0",1200, 8, "None", "One", "None", 1000, "None", "None", [252,82,48], False)
    # end: URCap Program Node
    $ 284 "Wait: 0.5"
    sleep(0.5)
    $ 285 "Set DO[0]=Off"
    set_standard_digital_out(0, False)
    $ 286 "MoveL"
    $ 287 "p4" "breakAfter"
    movel(p4, a=0.01, v=0.12)
    # begin: URCap Program Node
    #   Source: WireTank Serial, 4.9.0, WireTank, LLC
    #   Type: WireTank Serial
    $ 288 "Serial Bridge uR1"
    SerialResponse = WTSerialBridge.send_command("/dev/ttyUSB0",1200, 8, "None", "One", "None", 1000, "None", "None", [252,82,49], False)
    # end: URCap Program Node
    # begin: URCap Program Node
    #   Source: WireTank Serial, 4.9.0, WireTank, LLC
    #   Type: WireTank Serial
    $ 289 "Serial Bridge uR1"
    SerialResponse = WTSerialBridge.send_command("/dev/ttyUSB0",1200, 8, "None", "One", "None", 1000, "None", "None", [252,82,49], False)
    # end: URCap Program Node
    $ 290 "Wait: 1.0"
    sleep(1.0)
    $ 292 "Set DO[0]=On"
    set_standard_digital_out(0, True)
    $ 293 "MoveL"
    $ 294 "p5" "breakAfter"
    movel(p5, a=0.1, v=0.01)
    # begin: URCap Program Node
    #   Source: WireTank Serial, 4.9.0, WireTank, LLC
    #   Type: WireTank Serial
    $ 295 "Serial Bridge uR0"
    SerialResponse = WTSerialBridge.send_command("/dev/ttyUSB0",1200, 8, "None", "One", "None", 1000, "None", "None", [252,82,48], False)
    # end: URCap Program Node
    $ 296 "Wait: 2.0"
    sleep(2.0)
    $ 297 "Set DO[0]=Off"
    set_standard_digital_out(0, False)
    $ 298 "Comment"
    # Comment
    $ 299 "pret1≔p[p5[0]+.1,p5[1],p5[2],p5[3],p5[4],p5[5]]"
    global pret1=p[p5[0]+.1,p5[1],p5[2],p5[3],p5[4],p5[5]]
    $ 300 "p_1≔pathturn[4]"
    global p_1=pathturn[4]
    $ 301 "p_2≔pathturn[5]"
    global p_2=pathturn[5]
    $ 302 "p_3≔pathturn[6]"
    global p_3=pathturn[6]
    $ 303 "p_4≔pathturn[7]"
    global p_4=pathturn[7]
    $ 304 "p_5≔pathturn[8]"
    global p_5=pathturn[8]
    $ 305 "p_preheat≔p[p_3[0]+.01,p_3[1],p_3[2],p_3[3],p_3[4],p_3[5]]"
    global p_preheat=p[p_3[0]+.01,p_3[1],p_3[2],p_3[3],p_3[4],p_3[5]]
    $ 306 "p_pre_ret≔p[p_1[0]+.03,p_1[1]-.03,p_1[2],p_1[3],p_1[4],p_1[5]]"
    global p_pre_ret=p[p_1[0]+.03,p_1[1]-.03,p_1[2],p_1[3],p_1[4],p_1[5]]
    $ 307 "p_pre_ret2≔p[p_3[0]+.03,p_3[1],p_3[2],p_3[3],p_3[4],p_3[5]]"
    global p_pre_ret2=p[p_3[0]+.03,p_3[1],p_3[2],p_3[3],p_3[4],p_3[5]]
    $ 308 "MoveJ"
    $ 309 "pret1" "breakAfter"
    movej(pret1, a=1.3962634015954636, v=1.3962634015954636)
    $ 310 "Waypoint_28" "breakAfter"
    movej(get_inverse_kin(Waypoint_28_p, qnear=Waypoint_28_q), a=1.3962634015954636, v=1.3962634015954636)
    $ 311 "If liftcolumnz≠0.0"
    if (liftcolumnz != 0.0):
      # begin: URCap Program Node
      #   Source: MachineLogic for Universal Robots, 3.1.7, Vention Inc.
      #   Type: MachineLogic for Universal Robots
      $ 312 "MachineLogic Homing"
      while isVentionMovementBusyMachineMotion1==True:
      sleep(0.05)
      end
      if(isVentionMovementBusyMachineMotion1 == False):
      isVentionMovementBusyMachineMotion1 = True
      socket_send_string("estop/status;", "MachineMotion1")
      temp_estop_var_vention = socket_read_string("MachineMotion1",timeout=15)
      while(temp_estop_var_vention=="estop/status true"):
      if temp_estop_var_vention=="estop/status true":
      sendStringWithTimeout("estop/systemreset/request","Ack estop/systemreset/request;","MachineMotion1")
      end
      socket_send_string("estop/status;", "MachineMotion1")
      temp_estop_var_vention = socket_read_string("MachineMotion1",timeout=15)
      if temp_estop_var_vention=="estop/status true":
      popup("MachineMotion in estop, make sure you have all emergency modules released manually. If you continue the system will try to reset MachineMotion automatically.",blocking=True)
      end
      end
      else:
      popup("resource is being used already: MachineMotion1")
      halt
      end
      isVentionMovementBusyMachineMotion1 = True
      sendString("im_home_axis_1", "MachineMotion im_home_axis_1 = completed", "MachineMotion1")
      isVentionMovementBusyMachineMotion1 = False
      sendString("SET im_set_encoder_pos_aux_1 0.000", "Ack", "MachineMotion1")
      isVentionMovementBusyMachineMotion1 = False
      sleep(0.03)
      # end: URCap Program Node
    end
    $ 313 "'now go into the ccw weld position'"
    # 'now go into the ccw weld position'
    $ 314 "Waypoint_29" "breakAfter"
    movej(get_inverse_kin(Waypoint_29_p, qnear=Waypoint_29_q), a=1.3962634015954636, v=1.3962634015954636)
    $ 315 "Comment"
    # Comment
    $ 316 "Waypoint_30" "breakAfter"
    movej(get_inverse_kin(Waypoint_30_p, qnear=Waypoint_30_q), a=1.3962634015954636, v=1.3962634015954636)
    $ 317 "Waypoint_31" "breakAfter"
    movej(get_inverse_kin(Waypoint_31_p, qnear=Waypoint_31_q), a=1.3962634015954636, v=1.3962634015954636)
    $ 326 "MoveL"
    $ 327 "p_pre_ret" "breakAfter"
    movel(p_pre_ret, a=1.2, v=0.25)
    $ 328 "p_pre_ret2" "breakAfter"
    movel(p_pre_ret2, a=1.2, v=0.25)
    $ 329 "p_preheat" "breakAfter"
    movel(p_preheat, a=1.2, v=0.25)
    $ 330 "Wait: 6.0"
    sleep(6.0)
    $ 331 "MoveL"
    $ 332 "p_pre_ret2" "breakAfter"
    movel(p_pre_ret2, a=1.2, v=0.25)
    $ 333 "p_pre_ret" "breakAfter"
    movel(p_pre_ret, a=1.2, v=0.25)
    $ 334 "Set"
    set_tcp(p[0.00451,-0.328,0.105,1.2092,-1.2092,1.2092])
    $ 335 "MoveL"
    $ 336 "p_1" "breakAfter"
    movel(p_1, a=0.1, v=0.05)
    # begin: URCap Program Node
    #   Source: WireTank Serial, 4.9.0, WireTank, LLC
    #   Type: WireTank Serial
    $ 337 "Serial Bridge uR1"
    SerialResponse = WTSerialBridge.send_command("/dev/ttyUSB0",1200, 8, "None", "One", "None", 1000, "None", "None", [252,82,49], False)
    # end: URCap Program Node
    # begin: URCap Program Node
    #   Source: WireTank Serial, 4.9.0, WireTank, LLC
    #   Type: WireTank Serial
    $ 338 "Serial Bridge uR1"
    SerialResponse = WTSerialBridge.send_command("/dev/ttyUSB0",1200, 8, "None", "One", "None", 1000, "None", "None", [252,82,49], False)
    # end: URCap Program Node
    $ 339 "Wait: 1.0"
    sleep(1.0)
    $ 340 "Set DO[0]=On"
    set_standard_digital_out(0, True)
    $ 342 "Wait: 1.0"
    sleep(1.0)
    $ 343 "MoveL"
    $ 344 "p_2" "breakAfter"
    movel(p_2, a=1.2, v=0.01)
    $ 345 "MoveP"
    $ 346 "CircleMove"
    $ 347 "p_3" "noBreak"

    $ 348 "p_4" "breakAfter"
    movec(p_3, p_4, a=0.01, v=5.0E-4, r=0.0, mode=1)
    $ 349 "MoveL"
    $ 350 "p_5" "breakAfter"
    movel(p_5, a=1.2, v=0.012)
    # begin: URCap Program Node
    #   Source: WireTank Serial, 4.9.0, WireTank, LLC
    #   Type: WireTank Serial
    $ 351 "Serial Bridge uR0"
    SerialResponse = WTSerialBridge.send_command("/dev/ttyUSB0",1200, 8, "None", "One", "None", 1000, "None", "None", [252,82,48], False)
    # end: URCap Program Node
    $ 352 "Wait: 2.0"
    sleep(2.0)
    $ 353 "Set DO[0]=Off"
    set_standard_digital_out(0, False)
    $ 358 "MoveJ"
    $ 359 "Waypoint_32" "breakAfter"
    movej(get_inverse_kin(Waypoint_32_p, qnear=Waypoint_32_q), a=1.3962634015954636, v=1.0471975511965976)
    $ 360 "Waypoint_33" "breakAfter"
    movej(get_inverse_kin(Waypoint_33_p, qnear=Waypoint_33_q), a=1.3962634015954636, v=1.0471975511965976)
    $ 361 "Waypoint_73" "breakAfter"
    movej(get_inverse_kin(Waypoint_73_p, qnear=Waypoint_73_q), a=1.3962634015954636, v=1.0471975511965976)
    $ 362 "Comment"
    # Comment
    $ 363 "MoveJ"
    $ 364 "Waypoint_16" "breakAfter"
    movej(get_inverse_kin(Waypoint_16_p, qnear=Waypoint_16_q), a=1.3962634015954636, v=1.0471975511965976)
    $ 365 "Waypoint_17" "breakAfter"
    movej(get_inverse_kin(Waypoint_17_p, qnear=Waypoint_17_q), a=1.3962634015954636, v=1.0471975511965976)
    $ 366 "Waypoint_18" "breakAfter"
    movej(get_inverse_kin(Waypoint_18_p, qnear=Waypoint_18_q), a=1.3962634015954636, v=1.0471975511965976)
    $ 367 "Waypoint_38" "breakAfter"
    movej(get_inverse_kin(Waypoint_38_p, qnear=Waypoint_38_q), a=1.3962634015954636, v=1.0471975511965976)
    $ 368 "'above point is home'"
    # 'above point is home'
  end
  def Test_Teach_Position():
    $ 369 "Test_Teach_Position" "noBreak"
    $ 373 "MoveJ"
    $ 374 "Waypoint_40" "breakAfter"
    set_tcp(p[0.0,0.0,0.019,0.0,0.0,0.0])
    movej(get_inverse_kin(Waypoint_40_p, qnear=Waypoint_40_q), a=1.3962634015954636, v=1.0471975511965976)
    $ 375 "'above waypoint is home'"
    # 'above waypoint is home'
    $ 376 "Waypoint_2" "breakAfter"
    set_tcp(p[0.0,0.0,0.019,0.0,0.0,0.0])
    movej(get_inverse_kin(Waypoint_2_p, qnear=Waypoint_2_q), a=1.3962634015954636, v=1.0471975511965976)
    $ 377 "Set"
    set_tcp(p[1.4000000000000001E-4,-0.01751,0.284,0.0,0.0,0.0])
    $ 378 "freedrive_m_var≔ False "
    global freedrive_m_var=  False
    $ 379 "freedrive_m_var≔ True "
    global freedrive_m_var=  True
    $ 380 "Popup: Move the TCP to the top of the weld, then click 'Continue'"
    popup("Move the TCP to the top of the weld, then click 'Continue'", "Message", False, False, blocking=True)
    $ 381 "tcp_pose_top≔get_actual_tcp_pose()"
    global tcp_pose_top= get_actual_tcp_pose ()
    $ 382 "Popup: Move the TCP to the corner of the tank, then click 'Continue'"
    popup("Move the TCP to the corner of the tank, then click 'Continue'", "Message", False, False, blocking=True)
    $ 383 "tcp_pose≔get_actual_tcp_pose()"
    global tcp_pose= get_actual_tcp_pose ()
    $ 384 "freedrive_m_var≔ False "
    global freedrive_m_var=  False
    $ 385 "Wait: 0.25"
    sleep(0.25)
    $ 386 "sync()"
    sync()
  end
  def align_tcp_left():
    $ 387 "align_tcp_left" "noBreak"
    $ 388 "'this program aligns the tcp parallel to the y direction'"
    # 'this program aligns the tcp parallel to the y direction'
    $ 389 "cp≔get_actual_tcp_pose()"
    global cp= get_actual_tcp_pose ()
    $ 390 "aligned_y_pose≔p[cp[0],cp[1],cp[2],1.570796,0,0]"
    global aligned_y_pose=p[cp[0],cp[1],cp[2],1.570796,0,0]
    $ 391 "MoveJ"
    $ 392 "aligned_y_pose" "breakAfter"
    movej(aligned_y_pose, a=1.3962634015954636, v=1.0471975511965976)
  end
  def extrude_knife3():
    $ 393 "extrude_knife3" "noBreak"
    $ 394 "pre program stuff"
    $ 395 "Set"
    set_tcp(p[-0.011699999999999999,-0.328,0.105,1.2092,-1.2092,1.2092])
    $ 396 "ek_sp≔get_actual_tcp_pose()"
    global ek_sp= get_actual_tcp_pose ()
    $ 397 "MoveL"
    $ 398 "ek_sp" "breakAfter"
    movel(ek_sp, a=1.2, v=0.005)
    $ 399 "'list possible points'"
    # 'list possible points'
    $ 400 "robot 1 moves"
    $ 401 "If 1≟2"
    if (1 == 2):
      $ 402 "MoveJ"
      $ 403 "r1_ek_oldhome" "breakAfter"
      movej(get_inverse_kin(r1_ek_oldhome_p, qnear=r1_ek_oldhome_q), a=1.3962634015954636, v=1.0471975511965976)
      $ 404 "r1_ek_extrude" "breakAfter"
      movej(get_inverse_kin(r1_ek_extrude_p, qnear=r1_ek_extrude_q), a=1.3962634015954636, v=1.0471975511965976)
      $ 405 "r1_ek_front" "breakAfter"
      movej(get_inverse_kin(r1_ek_front_p, qnear=r1_ek_front_q), a=1.3962634015954636, v=1.0471975511965976)
      $ 406 "r1_ek_middle" "breakAfter"
      movej(get_inverse_kin(r1_ek_middle_p, qnear=r1_ek_middle_q), a=1.3962634015954636, v=1.0471975511965976)
      $ 407 "r1_ek_middle2" "breakAfter"
      movej(get_inverse_kin(r1_ek_middle2_p, qnear=r1_ek_middle2_q), a=1.3962634015954636, v=1.0471975511965976)
      $ 408 "r1_ek_bottom" "breakAfter"
      movej(get_inverse_kin(r1_ek_bottom_p, qnear=r1_ek_bottom_q), a=1.3962634015954636, v=1.0471975511965976)
      $ 409 "r1_ek_end" "breakAfter"
      movej(get_inverse_kin(r1_ek_end_p, qnear=r1_ek_end_q), a=1.3962634015954636, v=1.0471975511965976)
    end
    $ 410 "robot 2 moves"
    $ 411 "If 1≟2"
    if (1 == 2):
      $ 412 "MoveJ"
      $ 413 "r2_ek_oldhome" "breakAfter"
      movej(get_inverse_kin(r2_ek_oldhome_p, qnear=r2_ek_oldhome_q), a=1.3962634015954636, v=1.0471975511965976)
      $ 415 "r2_ek_extrude" "breakAfter"
      movej(get_inverse_kin(r2_ek_extrude_p, qnear=r2_ek_extrude_q), a=1.3962634015954636, v=1.0471975511965976)
      $ 416 "r2_ek_front" "breakAfter"
      movej(get_inverse_kin(r2_ek_front_p, qnear=r2_ek_front_q), a=1.3962634015954636, v=1.0471975511965976)
      $ 417 "r2_ek_middle" "breakAfter"
      movej(get_inverse_kin(r2_ek_middle_p, qnear=r2_ek_middle_q), a=1.3962634015954636, v=1.0471975511965976)
      $ 418 "r2_ek_bottom" "breakAfter"
      movej(get_inverse_kin(r2_ek_bottom_p, qnear=r2_ek_bottom_q), a=1.3962634015954636, v=1.0471975511965976)
      $ 419 "r2_ek_end" "breakAfter"
      movej(get_inverse_kin(r2_ek_end_p, qnear=r2_ek_end_q), a=1.3962634015954636, v=1.0471975511965976)
    end
    $ 420 "'detemine correct points for which robot'"
    # 'detemine correct points for which robot'
    $ 421 "If robot_number≟1"
    if (robot_number == 1):
      $ 422 "robot1 positions"
      $ 423 "ek_oldhome≔r1_ek_oldhome_p"
      global ek_oldhome=r1_ek_oldhome_p
      $ 424 "ek_extrude≔r1_ek_extrude_p"
      global ek_extrude=r1_ek_extrude_p
      $ 425 "ek_front≔r1_ek_front_p"
      global ek_front=r1_ek_front_p
      $ 426 "ek_middle≔r1_ek_middle_p"
      global ek_middle=r1_ek_middle_p
      $ 427 "ek_middle2≔r1_ek_middle2_p"
      global ek_middle2=r1_ek_middle2_p
      $ 428 "ek_bottom≔r1_ek_bottom_p"
      global ek_bottom=r1_ek_bottom_p
      $ 429 "ek_end≔r1_ek_end_q"
      global ek_end=r1_ek_end_q
    else:
      $ 430 "ElseIf robot_number≟2"
      if (robot_number == 2):
        $ 431 "robot1 positions"
        $ 432 "ek_oldhome≔r2_ek_oldhome_p"
        global ek_oldhome=r2_ek_oldhome_p
        $ 433 "ek_extrude≔r2_ek_extrude_p"
        global ek_extrude=r2_ek_extrude_p
        $ 434 "ek_front≔r2_ek_front_p"
        global ek_front=r2_ek_front_p
        $ 435 "ek_middle≔r2_ek_middle_p"
        global ek_middle=r2_ek_middle_p
        $ 436 "ek_middle2≔r2_ek_middle_p"
        global ek_middle2=r2_ek_middle_p
        $ 437 "ek_bottom≔r2_ek_bottom_p"
        global ek_bottom=r2_ek_bottom_p
        $ 438 "ek_end≔r2_ek_end_q"
        global ek_end=r2_ek_end_q
      end
    end
    $ 439 "'start of program'"
    # 'start of program'
    $ 441 "Set"
    set_tcp(p[-0.011699999999999999,-0.328,0.105,1.2092,-1.2092,1.2092])
    $ 442 "MoveJ"
    $ 444 "ek_oldhome" "breakAfter"
    movej(ek_oldhome, a=1.3962634015954636, v=1.0471975511965976)
    $ 445 "'above waypoint is home'"
    # 'above waypoint is home'
    $ 446 "'move above bucket'"
    # 'move above bucket'
    $ 447 "MoveJ"
    $ 449 "ek_extrude" "breakAfter"
    movej(ek_extrude, a=1.3962634015954636, v=1.0471975511965976)
    $ 450 "'extrude out a foot'"
    # 'extrude out a foot'
    # begin: URCap Program Node
    #   Source: WireTank Serial, 4.9.0, WireTank, LLC
    #   Type: WireTank Serial
    $ 452 "Serial Bridge uR1"
    SerialResponse = WTSerialBridge.send_command("/dev/ttyUSB0",1200, 8, "None", "One", "None", 1000, "None", "None", [252,82,49], False)
    # end: URCap Program Node
    $ 453 "Set DO[0]=On"
    set_standard_digital_out(0, True)
    $ 454 "Wait: 24.0"
    sleep(24.0)
    # begin: URCap Program Node
    #   Source: WireTank Serial, 4.9.0, WireTank, LLC
    #   Type: WireTank Serial
    $ 455 "Serial Bridge uR0"
    SerialResponse = WTSerialBridge.send_command("/dev/ttyUSB0",1200, 8, "None", "One", "None", 1000, "None", "None", [252,82,48], False)
    # end: URCap Program Node
    $ 456 "Wait: 1.0"
    sleep(1.0)
    $ 457 "Set DO[0]=Off"
    set_standard_digital_out(0, False)
    $ 458 "'slice'"
    # 'slice'
    $ 459 "MoveL"
    $ 465 "ek_front" "breakAfter"
    movel(ek_front, a=0.05, v=0.03)
    $ 466 "ek_middle" "breakAfter"
    movel(ek_middle, a=0.05, v=0.03)
    $ 467 "ek_middle2" "breakAfter"
    movel(ek_middle2, a=0.05, v=0.03)
    $ 468 "ek_bottom" "breakAfter"
    movel(ek_bottom, a=0.05, v=0.03)
    $ 469 "ek_end" "breakAfter"
    movel(ek_end, a=0.05, v=0.03)
    $ 470 "MoveJ"
    $ 472 "ek_oldhome" "breakAfter"
    movej(ek_oldhome, a=1.3962634015954636, v=1.0471975511965976)
    $ 473 "'above waypoint is home'"
    # 'above waypoint is home'
  end
  def align_tcp_forward():
    $ 475 "align_tcp_forward" "noBreak"
    $ 476 "'this program aligns the tcp parallel to the y direction'"
    # 'this program aligns the tcp parallel to the y direction'
    $ 477 "cp≔get_actual_tcp_pose()"
    global cp= get_actual_tcp_pose ()
    $ 478 "aligned_y_pose≔p[cp[0],cp[1],cp[2],0,-1.570796,0]"
    global aligned_y_pose=p[cp[0],cp[1],cp[2],0,-1.570796,0]
    $ 479 "MoveJ"
    $ 480 "aligned_y_pose" "breakAfter"
    movej(aligned_y_pose, a=1.3962634015954636, v=1.0471975511965976)
  end
  def align_tcp_up():
    $ 481 "align_tcp_up" "noBreak"
    $ 482 "'this program aligns the tcp parallel to the y direction'"
    # 'this program aligns the tcp parallel to the y direction'
    $ 483 "cp≔get_actual_tcp_pose()"
    global cp= get_actual_tcp_pose ()
    $ 484 "aligned_y_pose≔p[cp[0],cp[1],cp[2],0,0,0]"
    global aligned_y_pose=p[cp[0],cp[1],cp[2],0,0,0]
    $ 485 "MoveJ"
    $ 486 "aligned_y_pose" "breakAfter"
    movej(aligned_y_pose, a=1.3962634015954636, v=1.0471975511965976)
  end
  def align_ready_for_welding():
    $ 487 "align_ready_for_welding" "noBreak"
    $ 488 "'this program takes the welder from home to a position alined ready for welding (vertically down)'"
    # 'this program takes the welder from home to a position alined ready for welding (vertically down)'
    $ 489 "MoveJ"
    $ 490 "oldhome" "breakAfter"
    movej(get_inverse_kin(oldhome_p, qnear=oldhome_q), a=1.3962634015954636, v=1.0471975511965976)
    $ 491 "Waypoint_34" "breakAfter"
    movej(get_inverse_kin(Waypoint_34_p, qnear=Waypoint_34_q), a=1.3962634015954636, v=1.0471975511965976)
    $ 492 "Waypoint_35" "breakAfter"
    movej(get_inverse_kin(Waypoint_35_p, qnear=Waypoint_35_q), a=1.3962634015954636, v=1.0471975511965976)
    $ 493 "Waypoint_36" "breakAfter"
    movej(get_inverse_kin(Waypoint_36_p, qnear=Waypoint_36_q), a=1.3962634015954636, v=1.0471975511965976)
  end
  def Corner_Homing_45():
    $ 494 "Corner_Homing_45" "noBreak"
    $ 495 "'Use this program when tool is already positioned close to corner at 45deg'"
    # 'Use this program when tool is already positioned close to corner at 45deg'
    $ 496 "'tool flange will seek all 3 sides. will save those 5 locs in p__'"
    # 'tool flange will seek all 3 sides. will save those 5 locs in p__'
    $ 497 "Set"
    set_tcp(p[1.4000000000000001E-4,-0.01751,0.284,0.0,0.0,0.0])
    $ 506 "Wait: 1.0"
    sleep(1.0)
    $ 507 "tp≔get_actual_tcp_pose()"
    global tp= get_actual_tcp_pose ()
    $ 511 "path_pre≔get_corner_homing_45_pathpoints(tp,tcp_pose_top)"
    global path_pre=get_corner_homing_45_pathpoints(tp,tcp_pose_top)
    $ 512 "ph1≔path_pre[0]"
    global ph1=path_pre[0]
    $ 513 "ph2≔path_pre[1]"
    global ph2=path_pre[1]
    $ 514 "ph3≔path_pre[2]"
    global ph3=path_pre[2]
    $ 515 "ph4≔path_pre[3]"
    global ph4=path_pre[3]
    $ 516 "ph5≔path_pre[4]"
    global ph5=path_pre[4]
    $ 517 "ph6≔path_pre[5]"
    global ph6=path_pre[5]
    $ 518 "ph7≔path_pre[6]"
    global ph7=path_pre[6]
    $ 519 "ph2up≔path_pre[7]"
    global ph2up=path_pre[7]
    $ 520 "ph4up≔path_pre[8]"
    global ph4up=path_pre[8]
    $ 521 "MoveL"
    $ 522 "ph1" "breakAfter"
    movel(ph1, a=0.2, v=0.25)
    $ 523 "ph2" "breakAfter"
    movel(ph2, a=0.2, v=0.25)
    $ 524 "Wait: 0.5"
    sleep(0.5)
    $ 525 "MoveL"
    $ 526 "Direction: Base"
    global move_thread_flag_526=0
    thread move_thread_526():
      enter_critical
      move_thread_flag_526 = 1
      local towardsPos=calculate_point_to_move_towards(p[0.0,0.0,0.0,0.0,0.0,0.0], [-1,-1.0,0.0], 1000.0)
      movel(towardsPos, a=0.1, v=0.02)
      move_thread_flag_526 = 2
      exit_critical
    end
    move_thread_flag_526 = 0
    move_thread_han_526 = run move_thread_526()
    while (True):
      local targetTcpDirection=get_target_tcp_speed()
      local stepsToRetract=tool_contact(direction=targetTcpDirection)
      if (stepsToRetract > 0):
        kill move_thread_han_526
        stopl(3.0)
        local backTrackMovement=get_actual_joint_positions_history(stepsToRetract)
        local contactPose=get_forward_kin(backTrackMovement)
        local posDir=[targetTcpDirection[0],targetTcpDirection[1],targetTcpDirection[2]]
        local retractTo=contactPose
        if (norm(posDir) > 1e-6):
          local normalizedPosDir=normalize(posDir)
          local additionalRetraction=p[normalizedPosDir[0] * 0.0, normalizedPosDir[1] * 0.0, normalizedPosDir[2] * 0.0, 0, 0, 0]
          retractTo = pose_sub(contactPose, additionalRetraction)
        end
        movel(retractTo, a=3.0, v=0.1)
        $ 527 "Until (tool_contact_detection)"
        break
      end
      sync()
    end
    $ 528 "p11≔get_actual_tcp_pose()"
    global p11= get_actual_tcp_pose ()
    $ 529 "MoveJ"
    $ 530 "ph2" "breakAfter"
    movej(ph2, a=1.3962634015954636, v=1.0471975511965976)
    $ 531 "ph2up" "breakAfter"
    movej(ph2up, a=1.3962634015954636, v=1.0471975511965976)
    $ 532 "Wait: 0.5"
    sleep(0.5)
    $ 533 "MoveL"
    $ 534 "Direction: Base"
    global move_thread_flag_534=0
    thread move_thread_534():
      enter_critical
      move_thread_flag_534 = 1
      local towardsPos=calculate_point_to_move_towards(p[0.0,0.0,0.0,0.0,0.0,0.0], [-1,-1.0,0.0], 1000.0)
      movel(towardsPos, a=0.1, v=0.02)
      move_thread_flag_534 = 2
      exit_critical
    end
    move_thread_flag_534 = 0
    move_thread_han_534 = run move_thread_534()
    while (True):
      local targetTcpDirection=get_target_tcp_speed()
      local stepsToRetract=tool_contact(direction=targetTcpDirection)
      if (stepsToRetract > 0):
        kill move_thread_han_534
        stopl(3.0)
        local backTrackMovement=get_actual_joint_positions_history(stepsToRetract)
        local contactPose=get_forward_kin(backTrackMovement)
        local posDir=[targetTcpDirection[0],targetTcpDirection[1],targetTcpDirection[2]]
        local retractTo=contactPose
        if (norm(posDir) > 1e-6):
          local normalizedPosDir=normalize(posDir)
          local additionalRetraction=p[normalizedPosDir[0] * 0.0, normalizedPosDir[1] * 0.0, normalizedPosDir[2] * 0.0, 0, 0, 0]
          retractTo = pose_sub(contactPose, additionalRetraction)
        end
        movel(retractTo, a=3.0, v=0.1)
        $ 535 "Until (tool_contact_detection)"
        break
      end
      sync()
    end
    $ 536 "p13≔get_actual_tcp_pose()"
    global p13= get_actual_tcp_pose ()
    $ 537 "MoveJ"
    $ 538 "ph2up" "breakAfter"
    movej(ph2up, a=1.3962634015954636, v=1.0471975511965976)
    $ 539 "ph3" "breakAfter"
    movej(ph3, a=1.3962634015954636, v=1.0471975511965976)
    $ 540 "Wait: 0.5"
    sleep(0.5)
    $ 541 "MoveL"
    $ 542 "Direction: Base"
    global move_thread_flag_542=0
    thread move_thread_542():
      enter_critical
      move_thread_flag_542 = 1
      local towardsPos=calculate_point_to_move_towards(p[0.0,0.0,0.0,0.0,0.0,0.0], [-1,-1.0,0.0], 1000.0)
      movel(towardsPos, a=0.1, v=0.02)
      move_thread_flag_542 = 2
      exit_critical
    end
    move_thread_flag_542 = 0
    move_thread_han_542 = run move_thread_542()
    while (True):
      local targetTcpDirection=get_target_tcp_speed()
      local stepsToRetract=tool_contact(direction=targetTcpDirection)
      if (stepsToRetract > 0):
        kill move_thread_han_542
        stopl(3.0)
        local backTrackMovement=get_actual_joint_positions_history(stepsToRetract)
        local contactPose=get_forward_kin(backTrackMovement)
        local posDir=[targetTcpDirection[0],targetTcpDirection[1],targetTcpDirection[2]]
        local retractTo=contactPose
        if (norm(posDir) > 1e-6):
          local normalizedPosDir=normalize(posDir)
          local additionalRetraction=p[normalizedPosDir[0] * 0.0, normalizedPosDir[1] * 0.0, normalizedPosDir[2] * 0.0, 0, 0, 0]
          retractTo = pose_sub(contactPose, additionalRetraction)
        end
        movel(retractTo, a=3.0, v=0.1)
        $ 543 "Until (tool_contact_detection)"
        break
      end
      sync()
    end
    $ 544 "p12≔get_actual_tcp_pose()"
    global p12= get_actual_tcp_pose ()
    $ 548 "MoveL"
    $ 549 "ph3" "breakAfter"
    movel(ph3, a=1.2, v=0.25)
    $ 550 "ph1" "breakAfter"
    movel(ph1, a=1.2, v=0.25)
    $ 555 "MoveL"
    $ 556 "ph4" "breakAfter"
    movel(ph4, a=1.2, v=0.25)
    $ 557 "Wait: 0.5"
    sleep(0.5)
    $ 558 "MoveL"
    $ 559 "Direction: Base"
    global move_thread_flag_559=0
    thread move_thread_559():
      enter_critical
      move_thread_flag_559 = 1
      local towardsPos=calculate_point_to_move_towards(p[0.0,0.0,0.0,0.0,0.0,0.0], [-1.0,1.0,0.0], 1000.0)
      movel(towardsPos, a=0.1, v=0.02)
      move_thread_flag_559 = 2
      exit_critical
    end
    move_thread_flag_559 = 0
    move_thread_han_559 = run move_thread_559()
    while (True):
      local targetTcpDirection=get_target_tcp_speed()
      local stepsToRetract=tool_contact(direction=targetTcpDirection)
      if (stepsToRetract > 0):
        kill move_thread_han_559
        stopl(3.0)
        local backTrackMovement=get_actual_joint_positions_history(stepsToRetract)
        local contactPose=get_forward_kin(backTrackMovement)
        local posDir=[targetTcpDirection[0],targetTcpDirection[1],targetTcpDirection[2]]
        local retractTo=contactPose
        if (norm(posDir) > 1e-6):
          local normalizedPosDir=normalize(posDir)
          local additionalRetraction=p[normalizedPosDir[0] * 0.0, normalizedPosDir[1] * 0.0, normalizedPosDir[2] * 0.0, 0, 0, 0]
          retractTo = pose_sub(contactPose, additionalRetraction)
        end
        movel(retractTo, a=3.0, v=0.1)
        $ 560 "Until (tool_contact_detection)"
        break
      end
      sync()
    end
    $ 561 "p21≔get_actual_tcp_pose()"
    global p21= get_actual_tcp_pose ()
    $ 562 "MoveL"
    $ 563 "ph4" "breakAfter"
    movel(ph4, a=1.2, v=0.25)
    $ 564 "ph4up" "breakAfter"
    movel(ph4up, a=1.2, v=0.25)
    $ 565 "Wait: 0.5"
    sleep(0.5)
    $ 566 "MoveL"
    $ 567 "Direction: Base"
    global move_thread_flag_567=0
    thread move_thread_567():
      enter_critical
      move_thread_flag_567 = 1
      local towardsPos=calculate_point_to_move_towards(p[0.0,0.0,0.0,0.0,0.0,0.0], [-1.0,1.0,0.0], 1000.0)
      movel(towardsPos, a=0.1, v=0.02)
      move_thread_flag_567 = 2
      exit_critical
    end
    move_thread_flag_567 = 0
    move_thread_han_567 = run move_thread_567()
    while (True):
      local targetTcpDirection=get_target_tcp_speed()
      local stepsToRetract=tool_contact(direction=targetTcpDirection)
      if (stepsToRetract > 0):
        kill move_thread_han_567
        stopl(3.0)
        local backTrackMovement=get_actual_joint_positions_history(stepsToRetract)
        local contactPose=get_forward_kin(backTrackMovement)
        local posDir=[targetTcpDirection[0],targetTcpDirection[1],targetTcpDirection[2]]
        local retractTo=contactPose
        if (norm(posDir) > 1e-6):
          local normalizedPosDir=normalize(posDir)
          local additionalRetraction=p[normalizedPosDir[0] * 0.0, normalizedPosDir[1] * 0.0, normalizedPosDir[2] * 0.0, 0, 0, 0]
          retractTo = pose_sub(contactPose, additionalRetraction)
        end
        movel(retractTo, a=3.0, v=0.1)
        $ 568 "Until (tool_contact_detection)"
        break
      end
      sync()
    end
    $ 569 "p23≔get_actual_tcp_pose()"
    global p23= get_actual_tcp_pose ()
    $ 570 "MoveL"
    $ 571 "ph4up" "breakAfter"
    movel(ph4up, a=1.2, v=0.25)
    $ 572 "ph5" "breakAfter"
    movel(ph5, a=1.2, v=0.25)
    $ 573 "Wait: 0.5"
    sleep(0.5)
    $ 574 "MoveL"
    $ 575 "Direction: Base"
    global move_thread_flag_575=0
    thread move_thread_575():
      enter_critical
      move_thread_flag_575 = 1
      local towardsPos=calculate_point_to_move_towards(p[0.0,0.0,0.0,0.0,0.0,0.0], [-1.0,1.0,0.0], 1000.0)
      movel(towardsPos, a=0.1, v=0.02)
      move_thread_flag_575 = 2
      exit_critical
    end
    move_thread_flag_575 = 0
    move_thread_han_575 = run move_thread_575()
    while (True):
      local targetTcpDirection=get_target_tcp_speed()
      local stepsToRetract=tool_contact(direction=targetTcpDirection)
      if (stepsToRetract > 0):
        kill move_thread_han_575
        stopl(3.0)
        local backTrackMovement=get_actual_joint_positions_history(stepsToRetract)
        local contactPose=get_forward_kin(backTrackMovement)
        local posDir=[targetTcpDirection[0],targetTcpDirection[1],targetTcpDirection[2]]
        local retractTo=contactPose
        if (norm(posDir) > 1e-6):
          local normalizedPosDir=normalize(posDir)
          local additionalRetraction=p[normalizedPosDir[0] * 0.0, normalizedPosDir[1] * 0.0, normalizedPosDir[2] * 0.0, 0, 0, 0]
          retractTo = pose_sub(contactPose, additionalRetraction)
        end
        movel(retractTo, a=3.0, v=0.1)
        $ 576 "Until (tool_contact_detection)"
        break
      end
      sync()
    end
    $ 577 "p22≔get_actual_tcp_pose()"
    global p22= get_actual_tcp_pose ()
    $ 588 "MoveJ"
    $ 589 "ph5" "breakAfter"
    movej(ph5, a=1.3962634015954636, v=1.0471975511965976)
    $ 590 "MoveL"
    $ 591 "ph4" "breakAfter"
    movel(ph4, a=1.2, v=0.25)
    $ 592 "ph1" "breakAfter"
    movel(ph1, a=1.2, v=0.25)
    $ 593 "MoveJ"
    $ 594 "Waypoint_4" "breakAfter"
    movej(get_inverse_kin(Waypoint_4_p, qnear=Waypoint_4_q), a=1.3962634015954636, v=1.0471975511965976)
    $ 595 "Waypoint_13" "breakAfter"
    movej(get_inverse_kin(Waypoint_13_p, qnear=Waypoint_13_q), a=1.3962634015954636, v=1.0471975511965976)
    $ 596 "Waypoint_1" "breakAfter"
    movej(get_inverse_kin(Waypoint_1_p, qnear=Waypoint_1_q), a=1.3962634015954636, v=1.0471975511965976)
    $ 597 "ph6" "breakAfter"
    movej(ph6, a=1.3962634015954636, v=1.0471975511965976)
    $ 598 "ph7" "breakAfter"
    movej(ph7, a=1.3962634015954636, v=1.0471975511965976)
    $ 599 "Wait: 1.0"
    sleep(1.0)
    $ 603 "MoveL"
    $ 604 "Direction: Base Z+"
    global move_thread_flag_604=0
    thread move_thread_604():
      enter_critical
      move_thread_flag_604 = 1
      local towardsPos=calculate_point_to_move_towards(p[0.0,0.0,0.0,0.0,0.0,0.0], [0.0,0.0,1.0], 1000.0)
      movel(towardsPos, a=0.1, v=0.02)
      move_thread_flag_604 = 2
      exit_critical
    end
    move_thread_flag_604 = 0
    move_thread_han_604 = run move_thread_604()
    while (True):
      local targetTcpDirection=get_target_tcp_speed()
      local stepsToRetract=tool_contact(direction=targetTcpDirection)
      if (stepsToRetract > 0):
        kill move_thread_han_604
        stopl(3.0)
        local backTrackMovement=get_actual_joint_positions_history(stepsToRetract)
        local contactPose=get_forward_kin(backTrackMovement)
        local posDir=[targetTcpDirection[0],targetTcpDirection[1],targetTcpDirection[2]]
        local retractTo=contactPose
        if (norm(posDir) > 1e-6):
          local normalizedPosDir=normalize(posDir)
          local additionalRetraction=p[normalizedPosDir[0] * 0.0, normalizedPosDir[1] * 0.0, normalizedPosDir[2] * 0.0, 0, 0, 0]
          retractTo = pose_sub(contactPose, additionalRetraction)
        end
        movel(retractTo, a=3.0, v=0.1)
        $ 605 "Until (tool_contact_detection)"
        break
      end
      sync()
    end
    $ 606 "p3≔get_actual_tcp_pose()"
    global p3= get_actual_tcp_pose ()
    $ 607 "MoveJ"
    $ 608 "ph7" "breakAfter"
    movej(ph7, a=1.3962634015954636, v=1.0471975511965976)
    $ 609 "ph6" "breakAfter"
    movej(ph6, a=1.3962634015954636, v=1.0471975511965976)
    $ 610 "Waypoint_14" "breakAfter"
    movej(get_inverse_kin(Waypoint_14_p, qnear=Waypoint_14_q), a=1.3962634015954636, v=1.0471975511965976)
    $ 611 "Waypoint_4" "breakAfter"
    movej(get_inverse_kin(Waypoint_4_p, qnear=Waypoint_4_q), a=1.3962634015954636, v=1.0471975511965976)
    $ 612 "Waypoint_41" "breakAfter"
    movej(get_inverse_kin(Waypoint_41_p, qnear=Waypoint_41_q), a=1.3962634015954636, v=1.0471975511965976)
    $ 613 "'above waypoint is home'"
    # 'above waypoint is home'
    $ 615 "Comment"
    # Comment
    $ 616 "Comment"
    # Comment
    $ 617 "Comment"
    # Comment
    $ 618 "Comment"
    # Comment
    $ 619 "Comment"
    # Comment
    $ 620 "Comment"
    # Comment
  end
  $ 2 "BeforeStart"
  $ 3 "Safe Home Folder"
  $ 4 "'if robot is not at home, send it back to home safely'"
  # 'if robot is not at home, send it back to home safely'
  $ 5 "'make sure the tcp is welder'"
  # 'make sure the tcp is welder'
  $ 6 "Set"
  set_tcp(p[-0.011699999999999999,-0.328,0.105,1.2092,-1.2092,1.2092])
  $ 7 "sp≔get_actual_tcp_pose()"
  global sp= get_actual_tcp_pose ()
  $ 8 "MoveL"
  $ 9 "sp" "breakAfter"
  movel(sp, a=1.2, v=0.25)
  $ 10 "'if first move is to a variable, skip automove'"
  # 'if first move is to a variable, skip automove'
  $ 11 "'turn off welder'"
  # 'turn off welder'
  # begin: URCap Program Node
  #   Source: WireTank Serial, 4.9.0, WireTank, LLC
  #   Type: WireTank Serial
  $ 12 "Serial Bridge uR0"
  SerialResponse = WTSerialBridge.send_command("/dev/ttyUSB0",1200, 8, "None", "One", "None", 1000, "None", "None", [252,82,48], False)
  # end: URCap Program Node
  $ 13 "Set DO[0]=Off"
  set_standard_digital_out(0, False)
  $ 14 "jp≔get_actual_joint_positions()"
  global jp= get_actual_joint_positions ()
  $ 15 "If sp[0]>0.600"
  if (sp[0]>0.600):
    $ 16 "'if x > 600 then above then home'"
    # 'if x > 600 then above then home'
    $ 17 "MoveJ"
    $ 19 "Waypoint_76" "breakAfter"
    movej(get_inverse_kin(Waypoint_76_p, qnear=Waypoint_76_q), a=1.3962634015954636, v=1.0471975511965976)
    $ 20 "Home"
    movej([-3.266929759358355, -1.2139462677784536, 1.5878387874396154, 1.1069165929565088, -0.0023738326664366483, -1.7891447305770605], a=1.3962634015954636, v=1.0471975511965976)
  else:
    $ 21 "Else" "noBreak"
    $ 22 "Popup: retreating to home"
    popup("retreating to home", "Message", False, False, blocking=True)
    $ 23 "'for rules 2-8, finish with oldhome then above then home'"
    # 'for rules 2-8, finish with oldhome then above then home'
    $ 24 "If -1.74<jp[4] and jp[4]<1.05 and -1.74<jp[3] and jp[3]<1.74"
    if (-1.74<jp[4]  and  jp[4]<1.05  and  -1.74<jp[3]  and  jp[3]<1.74):
      $ 25 "'if oldhome, test teach, then go straight to oldhome'"
      # 'if oldhome, test teach, then go straight to oldhome'
    else:
      $ 26 "ElseIf sp[0]<-.5 and jp[3]>3.14 and -2.62<jp[4] and jp[4]<-0.87"
      if (sp[0]<-.5  and  jp[3]>3.14  and  -2.62<jp[4]  and  jp[4]<-0.87):
        $ 27 "'if left side weld approach, left weld approach in reverse'"
        # 'if left side weld approach, left weld approach in reverse'
        $ 28 "MoveJ"
        $ 29 "Waypoint_50" "breakAfter"
        movej(get_inverse_kin(Waypoint_50_p, qnear=Waypoint_50_q), a=1.3962634015954636, v=1.0471975511965976)
        $ 30 "Waypoint_51" "breakAfter"
        movej(get_inverse_kin(Waypoint_51_p, qnear=Waypoint_51_q), a=1.3962634015954636, v=1.0471975511965976)
        $ 31 "Waypoint_52" "breakAfter"
        movej(get_inverse_kin(Waypoint_52_p, qnear=Waypoint_52_q), a=1.3962634015954636, v=1.0471975511965976)
        $ 32 "Waypoint_53" "breakAfter"
        movej(get_inverse_kin(Waypoint_53_p, qnear=Waypoint_53_q), a=1.3962634015954636, v=1.0471975511965976)
      else:
        $ 33 "ElseIf sp[0]<0 and 0<jp[3] and jp[3]<1.74 and 0.87<jp[4] and jp[4]<2.62"
        if (sp[0]<0  and  0<jp[3]  and  jp[3]<1.74  and  0.87<jp[4]  and  jp[4]<2.62):
          $ 34 "'if right side around, move back then wapoint 24 then oldhome'"
          # 'if right side around, move back then wapoint 24 then oldhome'
          $ 35 "If sp[0]<-1.0"
          if (sp[0]<-1.0):
            $ 36 "xback≔p[-1.0,sp[1],sp[2],sp[3],sp[4],sp[5]]"
            global xback=p[-1.0,sp[1],sp[2],sp[3],sp[4],sp[5]]
            $ 37 "MoveJ"
            $ 38 "xback" "breakAfter"
            movej(xback, a=1.3962634015954636, v=1.0471975511965976)
          end
          $ 39 "MoveJ"
          $ 40 "Waypoint_54" "breakAfter"
          movej(get_inverse_kin(Waypoint_54_p, qnear=Waypoint_54_q), a=1.3962634015954636, v=1.0471975511965976)
        else:
          $ 41 "ElseIf jp[3]>2.62 and jp[4]<-3.84"
          if (jp[3]>2.62  and  jp[4]<-3.84):
            $ 42 "'if left side second half, then left weld ending sequence'"
            # 'if left side second half, then left weld ending sequence'
            $ 43 "If jp[5]<0.35"
            if (jp[5]<0.35):
              $ 44 "MoveJ"
              $ 45 "Waypoint_65" "breakAfter"
              movej(get_inverse_kin(Waypoint_65_p, qnear=Waypoint_65_q), a=1.3962634015954636, v=1.0471975511965976)
            end
            $ 46 "MoveJ"
            $ 51 "'above is testing, below is real'"
            # 'above is testing, below is real'
            $ 52 "Waypoint_55" "breakAfter"
            movej(get_inverse_kin(Waypoint_55_p, qnear=Waypoint_55_q), a=1.3962634015954636, v=1.0471975511965976)
            $ 54 "Waypoint_59" "breakAfter"
            movej(get_inverse_kin(Waypoint_59_p, qnear=Waypoint_59_q), t=2.0)
            $ 55 "Waypoint_71" "breakAfter"
            movej(get_inverse_kin(Waypoint_71_p, qnear=Waypoint_71_q), a=1.3962634015954636, v=1.0471975511965976)
            $ 56 "Waypoint_58" "breakAfter"
            movej(get_inverse_kin(Waypoint_58_p, qnear=Waypoint_58_q), a=1.3962634015954636, v=1.0471975511965976)
            $ 57 "Waypoint_56" "breakAfter"
            movej(get_inverse_kin(Waypoint_56_p, qnear=Waypoint_56_q), a=1.3962634015954636, v=1.0471975511965976)
            $ 58 "Waypoint_57" "breakAfter"
            movej(get_inverse_kin(Waypoint_57_p, qnear=Waypoint_57_q), a=1.3962634015954636, v=1.0471975511965976)
          else:
            $ 59 "ElseIf jp[3]<-2.09"
            if (jp[3]<-2.09):
              $ 60 "'bottom homing'"
              # 'bottom homing'
              $ 61 "MoveJ"
              $ 63 "Comment"
              # Comment
              $ 64 "If sp[0]<-0.95"
              if (sp[0]<-0.95):
                $ 65 "xback≔p[-0.95,sp[1],sp[2],sp[3],sp[4],sp[5]]"
                global xback=p[-0.95,sp[1],sp[2],sp[3],sp[4],sp[5]]
                $ 66 "MoveL"
                $ 67 "xback" "breakAfter"
                movel(xback, a=1.2, v=0.25)
              end
              $ 68 "Waypoint_67" "breakAfter"
              movej(get_inverse_kin(Waypoint_67_p, qnear=Waypoint_67_q), a=1.3962634015954636, v=1.0471975511965976)
            else:
              $ 69 "ElseIf jp[3]<0 and jp[4]<-3.14"
              if (jp[3]<0  and  jp[4]<-3.14):
                $ 70 "'if left side homing, special unspin'"
                # 'if left side homing, special unspin'
                $ 71 "MoveJ"
                $ 73 "Comment"
                # Comment
                $ 74 "Waypoint_69" "breakAfter"
                movej(get_inverse_kin(Waypoint_69_p, qnear=Waypoint_69_q), a=1.3962634015954636, v=1.0471975511965976)
                $ 75 "Waypoint_70" "breakAfter"
                movej(get_inverse_kin(Waypoint_70_p, qnear=Waypoint_70_q), a=1.3962634015954636, v=1.0471975511965976)
              else:
                $ 76 "ElseIf (sp[4]<-3 or sp[4]>3) and -0.02<sp[5] and sp[5]<0.02"
                if ((sp[4]<-3  or  sp[4]>3)  and  -0.02<sp[5]  and  sp[5]<0.02):
                  $ 77 "'go straight to home'"
                  # 'go straight to home'
                else:
                  $ 78 "ElseIf 2>1"
                  if (2>1):
                    $ 79 "'if none of the other options, then error continuously'"
                    # 'if none of the other options, then error continuously'
                    $ 80 "Loop 2>1"
                    while (2>1):
                      $ 81 "Popup: Unknown Position. Find Calvin for Assistance"
                      popup("Unknown Position. Find Calvin for Assistance", "Message", False, False, blocking=True)
                    end
                  end
                end
              end
            end
          end
        end
      end
    end
    $ 82 "'insert logic for how to get back to oldhome'"
    # 'insert logic for how to get back to oldhome'
    $ 83 "'finish with oldhome then above then home'"
    # 'finish with oldhome then above then home'
    $ 84 "MoveJ"
    $ 85 "Waypoint_49" "breakAfter"
    movej(get_inverse_kin(Waypoint_49_p, qnear=Waypoint_49_q), a=1.3962634015954636, v=1.0471975511965976)
    $ 87 "Waypoint_75" "breakAfter"
    movej(get_inverse_kin(Waypoint_75_p, qnear=Waypoint_75_q), a=1.3962634015954636, v=1.0471975511965976)
    $ 88 "Home"
    movej([-3.266929759358355, -1.2139462677784536, 1.5878387874396154, 1.1069165929565088, -0.0023738326664366483, -1.7891447305770605], a=1.3962634015954636, v=1.0471975511965976)
    # begin: URCap Program Node
    #   Source: MachineLogic for Universal Robots, 3.1.7, Vention Inc.
    #   Type: MachineLogic for Universal Robots
    $ 89 "MachineLogic Homing"
    while isVentionMovementBusyMachineMotion1==True:
    sleep(0.05)
    end
    if(isVentionMovementBusyMachineMotion1 == False):
    isVentionMovementBusyMachineMotion1 = True
    socket_send_string("estop/status;", "MachineMotion1")
    temp_estop_var_vention = socket_read_string("MachineMotion1",timeout=15)
    while(temp_estop_var_vention=="estop/status true"):
    if temp_estop_var_vention=="estop/status true":
    sendStringWithTimeout("estop/systemreset/request","Ack estop/systemreset/request;","MachineMotion1")
    end
    socket_send_string("estop/status;", "MachineMotion1")
    temp_estop_var_vention = socket_read_string("MachineMotion1",timeout=15)
    if temp_estop_var_vention=="estop/status true":
    popup("MachineMotion in estop, make sure you have all emergency modules released manually. If you continue the system will try to reset MachineMotion automatically.",blocking=True)
    end
    end
    else:
    popup("resource is being used already: MachineMotion1")
    halt
    end
    isVentionMovementBusyMachineMotion1 = True
    sendString("im_home_axis_1", "MachineMotion im_home_axis_1 = completed", "MachineMotion1")
    isVentionMovementBusyMachineMotion1 = False
    sendString("SET im_set_encoder_pos_aux_1 0.000", "Ack", "MachineMotion1")
    isVentionMovementBusyMachineMotion1 = False
    sleep(0.03)
    # end: URCap Program Node
  end
  $ 621 "Thread_1"
  thread Thread_1():
    $ 622 "Loop  True "
    while (  True  ):
      $ 623 "If freedrive_m_var≟ True "
      if (freedrive_m_var ==   True  ):
        $ 624 "freedrive_mode()"
        freedrive_mode()
        $ 625 "free_dr_already≔ True "
        global free_dr_already=  True
      else:
        $ 626 "Else" "noBreak"
        $ 627 "If free_dr_already"
        if (free_dr_already):
          $ 628 "end_freedrive_mode()"
          end_freedrive_mode()
        end
      end
      $ 629 "sync()"
      sync()
    end
  end
  threadId_Thread_1 = run Thread_1()
  $ 90 "Robot Program"
  $ 91 "'start of main program'"
  # 'start of main program'
  $ 92 "Set"
  set_tcp(p[-0.011699999999999999,-0.328,0.105,1.2092,-1.2092,1.2092])
  $ 93 "Home"
  movej([-3.266929759358355, -1.2139462677784536, 1.5878387874396154, 1.1069165929565088, -0.0023738326664366483, -1.7891447305770605], a=1.3962634015954636, v=1.0471975511965976)
  $ 94 "Script: common_math.script"
  # this file contains math equations and operations, not specific to any one feature

  # define pi
  pi = 3.1415926535

  # given 3 points, this finds the plane and its equation
  # rereturns ax + by + cz + d = 0 in a list of [a, b, c, d]
  def findplane(p11, p12, p13):
      # extract coordinates
      x1 = p11[0]
      y1 = p11[1]
      z1 = p11[2]
      x2 = p12[0]
      y2 = p12[1]
      z2 = p12[2]
      x3 = p13[0]
      y3 = p13[1]
      z3 = p13[2]
      # create vectors from the points
      v1x = x2-x1
      v1y = y2-y1
      v1z = z2-z1
      v2x = x3-x1
      v2y = y3-y1
      v2z = z3-z1
      #calculate the normal vector using the cross product
      nx = v1y*v2z - v1z*v2y # i component
      ny = v1z*v2x - v1x*v2z # j component
      nz = v1x*v2y - v1y*v2x # k component
      # calculate d in the plane equation
      d = -1 * (nx*x1 + ny*y1 + nz*z1)
      ret = [nx, ny, nz, d]
      return ret
  end

  # this function finds the intersection point between two lines in the xy plane
  # takes 4 arguments: m1, b1, m2, b2
  # returns a list of [x,y] (the point of intersection)
  def find_intersection(m1, b1, m2, b2):
    # m1x+b1 = m2x+b2
    # m1x - m2x = b2 - b1
    # x = (b2-b1) / (m1-m2)
    x = (b2-b1) / (m1-m2)
    y = m1 * x + b1
    ret = [x, y]
    return ret
  end

  # this function finds the distance between 2 points in 3d space
  # it takes 6 arguments: x1, y1, z1, x2, y2, z2
  # it returns a distance
  def distance_between(x1, y1, z1, x2, y2, z2):
    distsquared = (x2-x1)*(x2-x1)+(y2-y1)*(y2-y1)+(z2-z1)*(z2-z1)
    dist = sqrt(distsquared)
    return dist
  end

  # this function takes a point, a unit vector, and a distance, and adds the distance to the point in the direction of the unit vector (3d space)
  # it returns a point as a list of coordinates
  def add_vectordistance_to_point(xi, yi, zi, uvx, uvy, uvz, delta):
    xf = xi + uvx * delta
    yf = yi + uvy * delta
    zf = zi + uvz * delta
    ret = [xf, yf, zf]
    return ret
  end

  # this function takes two rotation matrices, and multiplies them together, returning one matrix.
  # all matrices are in the form of a list.
  # all matrix values have constant values (no variables)
  def multiply_matrix(matrix1, matrix2):
      # retrieve values
      a11 = matrix1[0]
      a12 = matrix1[1]
      a13 = matrix1[2]
      a21 = matrix1[3]
      a22 = matrix1[4]
      a23 = matrix1[5]
      a31 = matrix1[6]
      a32 = matrix1[7]
      a33 = matrix1[8]
      b11 = matrix2[0]
      b12 = matrix2[1]
      b13 = matrix2[2]
      b21 = matrix2[3]
      b22 = matrix2[4]
      b23 = matrix2[5]
      b31 = matrix2[6]
      b32 = matrix2[7]
      b33 = matrix2[8]
      #calculate c values
      c11 = a11*b11 + a12*b21 + a13*b31
      c12 = a11*b12 + a12*b22 + a13*b32
      c13 = a11*b13 + a12*b23 + a13*b33
      c21 = a21*b11 + a22*b21 + a23*b31
      c22 = a21*b12 + a22*b22 + a23*b32
      c23 = a21*b13 + a22*b23 + a23*b33
      c31 = a31*b11 + a32*b21 + a33*b31
      c32 = a31*b12 + a32*b22 + a33*b32
      c33 = a31*b13 + a32*b23 + a33*b33
      # return resulting matrix
      ret = [c11, c12, c13, c21, c22, c23, c31, c32, c33]
      return ret
  end

  # this function converts a matrix to axis angle representations
  # this matrix is usually a resulting matrix (result of matrix multiplication) in normal use, given as a list
  # returns a list of [rx,ry,rz]
  def convert_matrix_to_axang(matrix1):
      # retrieve values
      a11 = matrix1[0]
      a12 = matrix1[1]
      a13 = matrix1[2]
      a21 = matrix1[3]
      a22 = matrix1[4]
      a23 = matrix1[5]
      a31 = matrix1[6]
      a32 = matrix1[7]
      a33 = matrix1[8]

      # First Half: find the angle
      # find the trace
      # using the formula: trace = a11 + a22 + a33
      trace = a11 + a22 + a33
      # find the angle using the formula: trace(matrix) = 1 + 2 cos(angle)
      angle = acos((trace - 1.0)/2.0)

      # Second Half: calculate the rotation axis
      axisxraw = a32 - a23
      axisyraw = a13 - a31
      axiszraw = a21 - a12
      # normalize axis
      magnitude = sqrt(axisxraw*axisxraw + axisyraw*axisyraw + axiszraw*axiszraw)
      axisxunit = axisxraw / magnitude
      axisyunit = axisyraw / magnitude
      axiszunit = axiszraw / magnitude

      # combine axis and angle into rxryrz representation
      rxout = axisxunit * angle
      ryout = axisyunit * angle
      rzout = axiszunit * angle
      return [rxout, ryout, rzout]
  end

  # this function takes a rotation and calculates the corresponding rotation matrix
  # input is (axis, direction, angle in radians)
  # example is ("x", 1, pi/6) = a 30 degree turn around the x axis in the positive direction (right hand rule)
  # returns a matrix (a list of 9 values)
  def get_rotation_matrix_from_description(axis, direction, angle):
      # get the angle
      a = angle * direction
      # get the axis
      if axis == "x" or axis == "X":
          matrix = [1, 0, 0, 0, cos(a), -1 * sin(a), 0, sin(a), cos(a)]
          return matrix
      end
      if axis == "y" or axis == "Y":
          matrix = [cos(a), 0, sin(a), 0, 1, 0, -1*sin(a), 0, cos(a)]
          return matrix
      end
      if axis == "z" or axis == "Z":
          matrix = [cos(a), -1*sin(a), 0, sin(a), cos(a), 0, 0, 0, 1]
          return matrix
      end
      # bad
      popuptext = "Error in get_rotation_matrix_from_description. "
      # infinite loop
      while 1==1:
        popup(popuptext, title="Code Error",blocking=True)
      end
  end

  # given a round over distance (in mm), calculate (based on 90 degrees) the distance from corner (line intersection) to midpoint of arc
  # returns a value (in mm) that you need to move from line intersection to midpoint (actual distance will be this times sqrt(2))
  def calc_rod_midpoint_90deg(rod):
      # the factor is (1- 1/sqrt(2))
      factor = 0.292893
      ret = rod * factor
      return ret
  end

  def crossproduct(vec1, vec2):
      nx = vec1[1]*vec2[2] - vec1[2]*vec2[1]
      ny = vec1[2]*vec2[0] - vec1[0]*vec2[2]
      nz = vec1[0]*vec2[1] - vec1[1]*vec2[0]
      ret = [nx, ny, nz]
      return ret
  end

  # Section: headings, angles, slopes conversions

  # this function converts a heading (ccw radians from the positive x axis) into rxryrz to be put into a point p[]
  # this will point the gun in this heading with the bottom side of the gun facing up.
  # the values used in this program were calculated by doing rotation matrix math in the file on WI-CALVINB10 C. Documents. Theory for converting rotations into axis angle representations
  def convert_heading_to_axang(heading):
   axisxraw = -1 * sin(heading)
   axisyraw = cos(heading) + 1
   axiszraw = sin(heading)

   magnitude = sqrt(axisxraw*axisxraw + axisyraw*axisyraw + axiszraw*axiszraw)

   axisxunit = axisxraw / magnitude
   axisyunit = axisyraw / magnitude
   axiszunit = axiszraw / magnitude

   angle = acos( (cos(heading) - 1) / 2 )

   rxout = axisxunit * angle
   ryout = axisyunit * angle
   rzout = axiszunit * angle

   return [rxout, ryout, rzout]
  end

  # this function converts a heading (ccw radians from the positive x axis) into rxryrz to be put into a point p[]
  # this will point the gun in this heading with the preheat side of the gun tip facing up. Used for welding in a vertical path.
  # the values used in this program were calculated by doing rotation matrix math in the file on WI-CALVINB10 C. Documents. Theory for converting rotations into axis angle representations
  def convert_heading_to_axang_preheatup(heading):
   axisxraw = -sin(heading) + 1
   axisyraw = cos(heading)
   axiszraw = cos(heading)

   magnitude = sqrt(axisxraw*axisxraw + axisyraw*axisyraw + axiszraw*axiszraw)

   axisxunit = axisxraw / magnitude
   axisyunit = axisyraw / magnitude
   axiszunit = axiszraw / magnitude

   angle = acos( (-sin(heading) - 1) / 2 )

   rxout = axisxunit * angle
   ryout = axisyunit * angle
   rzout = axiszunit * angle

   return [rxout, ryout, rzout]
  end

  # this function converts a heading (ccw radians from the positive x axis) into rxryrz to be put into a point p[]
  # this will point the gun in this heading with the preheat side of the gun tip facing down. Used for welding in a vertical path downwards.
  # the values used in this program were calculated by doing rotation matrix math in the file on WI-CALVINB10 C. Documents. Theory for converting rotations into axis angle representations
  def convert_heading_to_axang_preheatdown(heading):
   axisxraw = -sin(heading) - 1
   axisyraw = cos(heading)
   axiszraw = -cos(heading)

   magnitude = sqrt(axisxraw*axisxraw + axisyraw*axisyraw + axiszraw*axiszraw)

   axisxunit = axisxraw / magnitude
   axisyunit = axisyraw / magnitude
   axiszunit = axiszraw / magnitude

   angle = acos( (sin(heading) - 1) / 2 )

   rxout = axisxunit * angle
   ryout = axisyunit * angle
   rzout = axiszunit * angle

   return [rxout, ryout, rzout]
  end

  # this function converts a heading (ccw radians from the positive x axis) into rxryrz to be put into a point p[]
  # this will point the gun in this heading with the preheat side of the gun tip facing right. Used for welding counterclockwise around the box.
  # the values used in this program were calculated by doing rotation matrix math in the file on WI-CALVINB10 C. Documents. Theory for converting rotations into axis angle representations
  def convert_heading_to_axang_ccw(heading):
   axisxraw = -sin(heading)
   axisyraw = cos(heading) - 1
   axiszraw = -sin(heading)

   magnitude = sqrt(axisxraw*axisxraw + axisyraw*axisyraw + axiszraw*axiszraw)

   axisxunit = axisxraw / magnitude
   axisyunit = axisyraw / magnitude
   axiszunit = axiszraw / magnitude

   angle = acos( (-cos(heading) - 1) / 2 )

   rxout = axisxunit * angle
   ryout = axisyunit * angle
   rzout = axiszunit * angle

   return [rxout, ryout, rzout]
  end

  # given a heading, (ccw from +x axis), find the mx+b slope
  # fails if exactly vertical
  def get_slope_from_heading(heading):
      return tan(heading)
  end

  # this function converts a unit vector to its heading angle ccw from x+ axis
  # takes uvx and uvy
  # returns heading in radians
  def convert_uv_to_heading(uvx, uvy):
    baseang = atan(uvy/uvx)
    if uvx < 0:
      ang = baseang + pi
    elif uvy < 0:
      ang = baseang + pi * 2
    else:
      ang = baseang
    end
    return ang
  end

  # this function finds the equation of a line, perpendicular to a given line, and going through a given point
  # takes 3 arguments: m (the original line's slope), x (point's x coord), y (point's y coord). the b of the original line is not needed
  # returns a list of [m,b] (the slope and intercept of the new line)
  def find_perpendicular_line(origm, x, y):
    m = (1/origm) * -1
    b = y - m*x
    ret = [m, b]
    return ret
  end

  # returns the absolute value of a number
  def absolute(x):
      ret = x
      if x < 0:
          ret = -1 * x
      end
      return ret
  end
  $ 95 "Script: common_io.script"
  # common_io.script
  # this file contains IO (input/output) commands, commonly used by robot programs
  # includes rs232 commands, lift column commands, and calls to native universal robots functions (like get_inverse_kin_has_solution())


  # Section: rs232 commands ###############################

  # this function sends a signal to turn extrusion on
  def turn_extrusion_on():
    # flush the channel
    resp0 = send_serial_signal(["u", "r", "?"])
    # send the signal
    resp1 = send_serial_signal(["u", "R", "1"])
    # if resp <> "uR1"
    if resp1 != [252,82,49]:
      # turn off extrusion and heating. inform calvin
      resp2 = send_serial_signal(["u", "R", "0"])
      resp3 = send_serial_signal(["u", "H", "0"])
      popuptext = "Error code encountered while trying to start extrusion. Find Calvin. "
      while 1==1:
        popup(popuptext, title="Extrusion Error Code",blocking=True)
        popup(resp1, blocking=True)
      end
    end
  end

  # this function sends a signal and receives a response
  # signal is a list of 3 strings, 1 character each. first is u. second is the next character. third is final character
  def send_serial_signal(signal):
    signal2char = signal[1]
    signal3char = signal[2]
    listsignal = [252, get_corr_number(signal2char), get_corr_number(signal3char)]
    resp1 = WTSerialBridge.send_command("/dev/ttyUSB0",1200, 8, "None", "One", "None", 1000, "None", "None", listsignal, True)
    return resp1
  end

  # this function converts a letter into its ascii number
  def get_corr_number(letter):
    if letter == "A":
      return 65
    elif letter == "H":
      return 72
    elif letter == "R":
      return 82
    elif letter == "M":
      return 77
    elif letter == "E":
      return 69
    elif letter == "a":
      return 97
    elif letter == "b":
      return 98
    elif letter == "h":
      return 104
    elif letter == "r":
      return 114
    elif letter == "s":
      return 115
    elif letter == "m":
      return 109
    elif letter == "0":
      return 48
    elif letter == "1":
      return 49
    elif letter == "2":
      return 50
    elif letter == "3":
      return 51
    elif letter == "4":
      return 52
    elif letter == "5":
      return 53
    elif letter == "6":
      return 54
    elif letter == "7":
      return 55
    elif letter == "8":
      return 56
    elif letter == "9":
      return 57
    elif letter == "?":
      return 63
    end
  end

  # this function checks whether the welder is in the ready state.
  # to be called at the beginning of Main Program
  def welder_state_ready():
    # flush the channel
    resp0 = send_serial_signal(["u", "s", "?"])
    # send the signal
    resp1 = send_serial_signal(["u", "s", "?"])
    # if resp1 == [252,115,49] (us1) then it is ready. otherwise, it is not
    if resp1 != [252,115,49]:
      popuptext = "Welder is not ready for extrusion. Follow the instructions to start heating welder. "
      while 1==1:
        popup(popuptext, title="Welder Not Ready",blocking=True)
      end
    end

  end


  # Section: lift column commands ##################################

  # initialize a lift column extension needed of 0.0
  global liftcolumnzneeded = 0.0 # set this variable in mm

